// TwinCAT 3 PLC project TcoDrivesBeckhoffTests
// Title: TcoDrivesBeckhoffTests
// Company: Vortex.Library
// Author: TcOpenGroup
// ProjectVersion: 0.6.0.913
// ProgramVersion: 3.1.4024.12
// libraries:
//   Tc2_EtherCAT, * (Beckhoff Automation GmbH)
//   Tc2_MC2, * (Beckhoff Automation GmbH)
//   Tc2_Standard, * (Beckhoff Automation GmbH)
//   Tc2_System, * (Beckhoff Automation GmbH)
//   Tc3_Module, * (Beckhoff Automation GmbH)
//   TcoCore, 0.6.0.913 (Vortex.Library)
//   TcoDrivesBeckhoff, 0.6.0.913 (Vortex.Library)
// project tree:
//   GVLs/ GVL.TcGVL
//   / PlcTask1.TcTTO
//   POUs/ MAIN.TcPOU
//   Tests/TcoContext/ Sequence1Task.TcPOU, SomeTestPositions.TcPOU, SomeTestMultiPositions.TcPOU, WpfContext.TcPOU
//   Tests/TcoContext/WrappedComponent/ WrappedComponentExample.TcPOU, WrappedComponentExample_Config.TcDUT, WrappedComponentExample_Control.TcDUT, WrappedComponentExample_Status.TcDUT, WrappedComponentsExample.TcDUT
//   Tests/TcoDriveSimple/ eTcoDriveSimpleTests.TcDUT, TcoDriveSimpleTestContext.TcPOU, TcoDriveSimpleTest.TcPOU
//   Tests/TcoSingleAxis/ eTcoSingleAxisTests.TcDUT, TcoSingleAxisContext.TcPOU, TcoSingleAxisTest.TcPOU
//   Tests/TcoMultiAxis/ eTcoMultiAxisTests.TcDUT, TcoMultiAxisContext.TcPOU, TcoMultiAxisTest.TcPOU
// (motion and I/O tree: see PLC project tcodrivesbeckhoff)
// real-time tasks:
//   TASK PlcTask: cycle T#10ms, priority 20, ADS port 350
//   TASK PlcTask1: cycle T#10ms, priority 1, ADS port 351
// variable links:
//   TcoDrivesBeckhoffTests/TcoDrivesBeckhoffTests Instance <-> Device 2 (EtherCAT)/Term 1 (EK1200)/Term 12 (EL1809)
//     PlcTask1 Inputs/GVL._calibrationCam <-> Channel 1/Input
//   TcoDrivesBeckhoffTests/TcoDrivesBeckhoffTests Instance <-> NC-Task 1 SAF/Axes/Axis 1
//     PlcTask1 Inputs/GVL.Axis1.NcToPlc <-> Outputs/ToPlc
//     PlcTask1 Outputs/GVL.Axis1.PlcToNc <-> Inputs/FromPlc
//   TcoDrivesBeckhoffTests/TcoDrivesBeckhoffTests Instance <-> NC-Task 1 SAF/Axes/Axis 2
//     PlcTask1 Inputs/GVL.Axis2.NcToPlc <-> Outputs/ToPlc
//     PlcTask1 Outputs/GVL.Axis2.PlcToNc <-> Inputs/FromPlc
//   TcoDrivesBeckhoffTests/TcoDrivesBeckhoffTests Instance <-> NC-Task 1 SAF/Axes/Axis 3
//     PlcTask1 Inputs/GVL.Axis3.NcToPlc <-> Outputs/ToPlc
//     PlcTask1 Outputs/GVL.Axis3.PlcToNc <-> Inputs/FromPlc
//   TcoDrivesBeckhoffTests/TcoDrivesBeckhoffTests Instance <-> NC-Task 1 SAF/Axes/Axis 4
//     PlcTask1 Inputs/GVL.Axis4.NcToPlc <-> Outputs/ToPlc
//     PlcTask1 Outputs/GVL.Axis4.PlcToNc <-> Inputs/FromPlc

CONFIGURATION TcoDrivesBeckhoffTests
    RESOURCE PLC ON TwinCAT3
        TASK PlcTask1(INTERVAL := T#10ms, PRIORITY := 1);
        PROGRAM MAIN WITH PlcTask1 : MAIN;
    END_RESOURCE
END_CONFIGURATION

// ---- Tests/TcoContext/WrappedComponent/WrappedComponentExample_Config.TcDUT
TYPE WrappedComponentExample_Config EXTENDS TcoCore.TcoStruct :
STRUCT
    VacuumReachedStabilisation : TIME := T#100MS;
    VacuumPushTime : TIME := T#100MS;
END_STRUCT
END_TYPE

// ---- Tests/TcoContext/WrappedComponent/WrappedComponentExample_Control.TcDUT
TYPE WrappedComponentExample_Control EXTENDS TcoCore.TcoStruct :
STRUCT
    Setpoint : INT;
END_STRUCT
END_TYPE

// ---- Tests/TcoContext/WrappedComponent/WrappedComponentExample_Status.TcDUT
TYPE WrappedComponentExample_Status EXTENDS TcoCore.TcoStruct :
STRUCT
    ProgressThrow : INT;
    ActionDescription : STRING;
END_STRUCT
END_TYPE

// ---- Tests/TcoContext/WrappedComponent/WrappedComponentsExample.TcDUT
TYPE WrappedComponentsExample EXTENDS TcoCore.TcoStruct :
STRUCT
    {attribute addProperty Name "Manipulator"}
    Manipulator : TcoDrivesBeckhoff.TcoMultiAxis(THISSTRUCT);
    {attribute addProperty Name "Axis"}
    Axis : TcoDrivesBeckhoff.TcoSingleAxis(THISSTRUCT);
    {attribute addProperty Name "Drive"}
    Drive : TcoDrivesBeckhoff.TcoDriveSimple(THISSTRUCT);
END_STRUCT
END_TYPE

// ---- Tests/TcoDriveSimple/eTcoDriveSimpleTests.TcDUT
{attribute 'qualified_only'}
{attribute 'strict'}
TYPE eTcoDriveSimpleTests :
(
    Restore := 1,
    CleanUp,
    Message,
    PowerDisable,
    PowerEnable,
    Reset,
    MoveRelativePositiveWithDisabledPositiveDirection,
    MoveRelativePositiveWithEnabledPositiveDirection,
    MoveRelativeNegativeWithDisabledNegativeDirection,
    MoveRelativeNegativeWithEnabledNegativeDirection,
    HommingDirect,
    MoveVelocityPositiveWithDisabledPositiveDirection,
    MoveVelocityPositiveWithEnabledPositiveDirection,
    Stop,
    MoveVelocityNegativeWithDisabledNegativeDirection,
    MoveVelocityNegativeWithEnabledNegativeDirection,
    MoveAbsoluteDisabled,
    MoveAbsoluteDisabledPositiveDirection,
    MoveAbsoluteEnabledPositiveDirection,
    MoveAbsoluteDisabledNegativeDirection,
    MoveAbsoluteEnabledNegativeDirection,
    Last
);
END_TYPE

// ---- Tests/TcoSingleAxis/eTcoSingleAxisTests.TcDUT
{attribute 'qualified_only'}
{attribute 'strict'}
TYPE eTcoSingleAxisTests :
(
    Restore := 1,
    CleanUp,
    Message,
    PowerDisable,
    PowerEnable,
    Reset,
    MoveRelativePositiveWithDisabledPositiveDirection,
    MoveRelativePositiveWithEnabledPositiveDirection,
    MoveRelativeNegativeWithDisabledNegativeDirection,
    MoveRelativeNegativeWithEnabledNegativeDirection,
    HommingDirect,
    MoveVelocityPositiveWithDisabledPositiveDirection,
    MoveVelocityPositiveWithEnabledPositiveDirection,
    Stop,
    MoveVelocityNegativeWithDisabledNegativeDirection,
    MoveVelocityNegativeWithEnabledNegativeDirection,
    MoveAbsoluteDisabled,
    MoveAbsoluteDisabledPositiveDirection,
    MoveAbsoluteEnabledPositiveDirection,
    MoveAbsoluteDisabledNegativeDirection,
    MoveAbsoluteEnabledNegativeDirection,
    MoveAbsoluteAxisDisabled,
    MoveAbsoluteAxisDisabledPositiveDirection,
    MoveAbsoluteAxisEnabledPositiveDirection,
    MoveAbsoluteAxisDisabledNegativeDirection,
    MoveAbsoluteAxisEnabledNegativeDirection,
    MoveRelativeAxisDisabled,
    MoveRelativeAxisDisabledPositiveDirection,
    MoveRelativeAxisEnabledPositiveDirection,
    MoveRelativeAxisDisabledNegativeDirection,
    MoveRelativeAxisEnabledNegativeDirection,
    Last
);
END_TYPE

// ---- Tests/TcoMultiAxis/eTcoMultiAxisTests.TcDUT
{attribute 'qualified_only'}
{attribute 'strict'}
TYPE eTcoMultiAxisTests :
(
    Restore := 1,
    CleanUp,
    Message,
    PowerDisable,
    PowerEnable,
    Reset,
    HommingDirect,
    Stop,
    MoveAbsoluteDisabled,
    MoveAbsoluteDisabledPositiveDirection,
    MoveAbsoluteEnabledPositiveDirection,
    MoveAbsoluteDisabledNegativeDirection,
    MoveAbsoluteEnabledNegativeDirection,
    MoveAbsoluteAxisDisabled,
    MoveAbsoluteAxisDisabledPositiveDirection,
    MoveAbsoluteAxisEnabledPositiveDirection,
    MoveAbsoluteAxisDisabledNegativeDirection,
    MoveAbsoluteAxisEnabledNegativeDirection,
    MoveAbsoluteAxisDisabledPositiveDirectionAxisDisabled,
    MoveAbsoluteAxisEnabledPositiveDirectionAxisDisabled,
    MoveAbsoluteAxisDisabledNegativeDirectionAxisDisabled,
    MoveAbsoluteAxisEnabledNegativeDirectionAxisDisabled,
    Last
);
END_TYPE

// ---- GVLs/GVL.TcGVL
{attribute 'qualified_only'}
VAR_GLOBAL
    SimpleAxis1 : TcoDrivesBeckhoff.TcoAxisRef;
    SimpleAxis2 : TcoDrivesBeckhoff.TcoAxisRef;
    SingleAxis : TcoDrivesBeckhoff.TcoAxisRef;
    Axis1 : TcoDrivesBeckhoff.TcoAxisRef;
    Axis2 : TcoDrivesBeckhoff.TcoAxisRef;
    Axis3 : TcoDrivesBeckhoff.TcoAxisRef;
    Axis4 : TcoDrivesBeckhoff.TcoAxisRef;
    _calibrationCam AT %I* : BOOL;
END_VAR

// ---- POUs/MAIN.TcPOU
PROGRAM MAIN
VAR
    _tcoDriveSimpleTestContext : TcoDriveSimpleTestContext;
    _tcoSingleAxisTestContext : TcoSingleAxisContext;
    _tcoMultiAxisTestContext : TcoMultiAxisContext;
    _wpfContext : WpfContext;
    _wpfContextCall : BOOL := FALSE;
    _singleAxisTestActive : BOOL;
    _multiAxisTestActive : BOOL;
END_VAR

IF _singleAxisTestActive THEN
    _tcoSingleAxisTestContext.ProbeRun();
ELSIF _multiAxisTestActive THEN
    _tcoMultiAxisTestContext.ProbeRun();
ELSE
    _tcoDriveSimpleTestContext.ProbeRun();
END_IF

IF _wpfContextCall THEN
    _wpfContext.Run();
END_IF

END_PROGRAM

// ---- Tests/TcoDriveSimple/TcoDriveSimpleTestContext.TcPOU
FUNCTION_BLOCK TcoDriveSimpleTestContext EXTENDS TcoCore._internals_TcoContext
VAR
    _sut : TcoDriveSimpleTest(THIS^);
    _callMyPlcInstance : BOOL := FALSE;
    _enable : BOOL;
    _enablePositive : BOOL;
    _enableNegative : BOOL;
    _calibrationCam : BOOL;
    _position : LREAL;
    _velocity : LREAL;
    _acceleration : LREAL;
    _deceleration : LREAL;
    _jerk : LREAL;
    _inString : STRING;
    _done : BOOL;
    _arranged : BOOL;
    _axisReferenceType : INT;
END_VAR

METHOD PROTECTED Main
_sut(inEnable := _enable,
    inEnablePositive := _enablePositive,
    inEnableNegative := _enableNegative,
    inCalibrationCam := _calibrationCam,
    inoAxisRef := GVL.Axis1);

CASE _testId OF
    eTcoDriveSimpleTests.Restore:
        _sut.Restore();
    eTcoDriveSimpleTests.CleanUp:
        _sut._messenger.Clear();
        {region "T003_Message"}
    eTcoDriveSimpleTests.Message:
        _sut.Messenger.Error(_inString);
        _done := _plcCycleCounter > 1;
        ProbeDoneWhen(_done);
        {endregion}
        {region "T004_PowerDisable"}
    eTcoDriveSimpleTests.PowerDisable:
        _enable := FALSE;
        _done := _sut._axisStatus.Disabled; // OR _plcCycleCounter > 1;
        ProbeDoneWhen(_done);
        {endregion}
        {region "T005_PowerEnable"}
    eTcoDriveSimpleTests.PowerEnable:
        _enable := TRUE;
        _done := _sut._axisStatus.Operational; // OR _plcCycleCounter > 15;
        ProbeDoneWhen(_done);
        {endregion}
        {region "T006_Reset"}
    eTcoDriveSimpleTests.Reset:
        IF NOT _arranged THEN
            _sut.MoveRelative(inDistance := 500,
                inVelocity := 50000000,
                inAcceleration := -1,
                inDeceleration := -1,
                inJerk := -1);

            IF _sut._axisStatus.Error THEN
                _arranged := true;
            END_IF

            RETURN;
        END_IF

        _sut.Reset();
        _done := _sut.ResetTask.Done OR _sut.ResetTask.Error; // OR _plcCycleCounter > 1;
        ProbeDoneWhen(_done);
        {endregion}
        {region "T007_MoveRelativePositiveWithDisabledPositiveDirection"}
    eTcoDriveSimpleTests.MoveRelativePositiveWithDisabledPositiveDirection:
        IF NOT _arranged THEN
            _enable := TRUE;
            _enablePositive := FALSE;
            _enableNegative := FALSE;

            IF _sut._axisStatus.Operational THEN
                _arranged := TRUE;
            END_IF

            RETURN;
        END_IF;

        _sut.MoveRelative(inDistance := _position,
            inVelocity := _velocity,
            inAcceleration := _acceleration,
            inDeceleration := _deceleration,
            inJerk := _jerk);

        _done := _sut.MoveRelativeTask.Done OR _sut.MoveRelativeTask.Error; // OR _sut._axisStatus.Error;// OR _plcCycleCounter > 5;
        ProbeDoneWhen(_done);
        {endregion}
        {region "T008_MoveRelativePositiveWithEnabledPositiveDirection"}
    eTcoDriveSimpleTests.MoveRelativePositiveWithEnabledPositiveDirection:
        IF NOT _arranged THEN
            _enable := TRUE;
            _enablePositive := TRUE;
            _enableNegative := FALSE;

            IF _sut._axisStatus.Operational THEN
                _arranged := TRUE;
            END_IF

            RETURN;
        END_IF;

        _sut.MoveRelative(inDistance := _position,
            inVelocity := _velocity,
            inAcceleration := _acceleration,
            inDeceleration := _deceleration,
            inJerk := _jerk);

        _done := _sut.MoveRelativeTask.Done OR _sut.MoveRelativeTask.Error; // OR  _plcCycleCounter > 1000;
        ProbeDoneWhen(_done);
        {endregion}
        {region "T009_MoveRelativeNegativeWithDisabledNegativeDirection"}
    eTcoDriveSimpleTests.MoveRelativeNegativeWithDisabledNegativeDirection:
        IF NOT _arranged THEN
            _enable := TRUE;
            _enablePositive := FALSE;
            _enableNegative := FALSE;

            IF _sut._axisStatus.Operational THEN
                _arranged := TRUE;
            END_IF

            RETURN;
        END_IF;

        _sut.MoveRelative(inDistance := _position,
            inVelocity := _velocity,
            inAcceleration := _acceleration,
            inDeceleration := _deceleration,
            inJerk := _jerk);

        _done := _sut.MoveRelativeTask.Done OR _sut.MoveRelativeTask.Error; // OR _sut._axisStatus.Error;// OR _plcCycleCounter > 5;
        ProbeDoneWhen(_done);
        {endregion}
        {region "T010_MoveRelativeNegativeWithEnabledNegativeDirection"}
    eTcoDriveSimpleTests.MoveRelativeNegativeWithEnabledNegativeDirection:
        IF NOT _arranged THEN
            _enable := TRUE;
            _enablePositive := TRUE;
            _enableNegative := TRUE;

            IF _sut._axisStatus.Operational THEN
                _arranged := TRUE;
            END_IF

            RETURN;
        END_IF;

        _sut.MoveRelative(inDistance := _position,
            inVelocity := _velocity,
            inAcceleration := _acceleration,
            inDeceleration := _deceleration,
            inJerk := _jerk);

        _done := _sut.MoveRelativeTask.Done OR _sut.MoveRelativeTask.Error; // OR  _plcCycleCounter > 1000;
        ProbeDoneWhen(_done);
        {endregion}
        {region "T011_HommingDirect"}
    eTcoDriveSimpleTests.HommingDirect:
        IF NOT _arranged THEN
            _enable := TRUE;
            _enablePositive := FALSE;
            _enableNegative := TRUE;

            IF _sut._axisStatus.Operational THEN
                _arranged := TRUE;
            END_IF

            RETURN;
        END_IF;

        _sut.Home(inPosition := _position,
            inHomingMode := TcoDrivesBeckhoff.eHomingMode.MC_Direct,
            inClearPositionLag := FALSE,
            inSearchDirection := TcoDrivesBeckhoff.eDirection.MC_Undefined_Direction,
            inSearchVelocity := _velocity,
            inSyncDirection := TcoDrivesBeckhoff.eDirection.MC_Undefined_Direction,
            inSyncVelocity := _velocity,
            inReferenceMode := TcoDrivesBeckhoff.eEncoderReferenceMode.ENCODERREFERENCEMODE_DEFAULT);

        _done := _sut.HomeTask.Done OR _sut.HomeTask.Error; //OR _plcCycleCounter > 1000;
        ProbeDoneWhen(_done);
        {endregion}
        {region "T012_MoveVelocityPositiveWithDisabledPositiveDirection"}
    eTcoDriveSimpleTests.MoveVelocityPositiveWithDisabledPositiveDirection:
        IF NOT _arranged THEN
            _enable := TRUE;
            _enablePositive := FALSE;
            _enableNegative := FALSE;

            IF _sut._axisStatus.Operational THEN
                _arranged := TRUE;
            END_IF

            RETURN;
        END_IF;

        _sut.MoveVelocity(inVelocity := _velocity,
            inAcceleration := _acceleration,
            inDeceleration := _deceleration,
            inJerk := _jerk,
            inDirection := TcoDrivesBeckhoff.eDirection.MC_Positive_Direction);

        _done := _sut.MoveVelocityTask.Done OR _sut.MoveVelocityTask.Error; // OR  _sut._axisStatus.Error;// OR _plcCycleCounter > 5;
        ProbeDoneWhen(_done);
        {endregion}
        {region "T013_MoveVelocityPositiveWithEnabledPositiveDirection"}
    eTcoDriveSimpleTests.MoveVelocityPositiveWithEnabledPositiveDirection:
        IF NOT _arranged THEN
            _enable := TRUE;
            _enablePositive := TRUE;
            _enableNegative := FALSE;

            IF _sut._axisStatus.Operational THEN
                _arranged := TRUE;
            END_IF

            RETURN;
        END_IF;

        _sut.MoveVelocity(inVelocity := _velocity,
            inAcceleration := _acceleration,
            inDeceleration := _deceleration,
            inJerk := _jerk,
            inDirection := TcoDrivesBeckhoff.eDirection.MC_Positive_Direction);

        _done := _sut.MoveVelocityTask.Done OR _sut.MoveVelocityTask.Error; // OR  _plcCycleCounter > 1000;
        ProbeDoneWhen(_done);
        {endregion}
        {region "T014_Stop"}
    eTcoDriveSimpleTests.Stop:
        IF NOT _arranged THEN
            _enable := TRUE;
            _enablePositive := TRUE;
            _enableNegative := TRUE;

            IF _sut._axisStatus.Operational THEN
                _arranged := TRUE;
            END_IF

            RETURN;
        END_IF;

        _sut.Stop(inDeceleration := _deceleration, inJerk := _jerk);
        _done := _sut.StopTask.Done OR _sut.StopTask.Error; // OR  _plcCycleCounter > 1000;
        ProbeDoneWhen(_done);
        {endregion}
        {region "T015_MoveVelocityNegativeWithDisabledNegativeDirection"}
    eTcoDriveSimpleTests.MoveVelocityNegativeWithDisabledNegativeDirection:
        IF NOT _arranged THEN
            _enable := TRUE;
            _enablePositive := FALSE;
            _enableNegative := FALSE;

            IF _sut._axisStatus.Operational THEN
                _arranged := TRUE;
            END_IF

            RETURN;
        END_IF;

        _sut.MoveVelocity(inVelocity := _velocity,
            inAcceleration := _acceleration,
            inDeceleration := _deceleration,
            inJerk := _jerk,
            inDirection := TcoDrivesBeckhoff.eDirection.MC_Negative_Direction);

        _done := _sut.MoveVelocityTask.Done OR _sut.MoveVelocityTask.Error; // OR  _sut._axisStatus.Error;// OR _plcCycleCounter > 5;
        ProbeDoneWhen(_done);
        {endregion}
        {region "T016_MoveVelocityNegativeWithEnabledNegativeDirection"}
    eTcoDriveSimpleTests.MoveVelocityNegativeWithEnabledNegativeDirection:
        IF NOT _arranged THEN
            _enable := TRUE;
            _enablePositive := FALSE;
            _enableNegative := TRUE;

            IF _sut._axisStatus.Operational THEN
                _arranged := TRUE;
            END_IF

            RETURN;
        END_IF;

        _sut.MoveVelocity(inVelocity := _velocity,
            inAcceleration := _acceleration,
            inDeceleration := _deceleration,
            inJerk := _jerk,
            inDirection := TcoDrivesBeckhoff.eDirection.MC_Negative_Direction);

        _done := _sut.MoveVelocityTask.Done OR _sut.MoveVelocityTask.Error; // OR  _plcCycleCounter > 1000;
        ProbeDoneWhen(_done);
        {endregion}
        {region "T017_MoveAbsoluteDisabled"}
    eTcoDriveSimpleTests.MoveAbsoluteDisabled:
        IF NOT _arranged THEN
            _enable := FALSE;
            _enablePositive := FALSE;
            _enableNegative := FALSE;
            _arranged := TRUE;
            RETURN;
        END_IF;

        _sut.MoveAbsolute(inPosition := _position,
            inVelocity := _velocity,
            inAcceleration := _acceleration,
            inDeceleration := _deceleration,
            inJerk := _jerk);

        _done := _sut.MoveAbsoluteTask.Done OR _sut.MoveAbsoluteTask.Error OR _plcCycleCounter > 10;
        ProbeDoneWhen(_done);
        {endregion}
        {region "T018_MoveAbsoluteDisabledPositiveDirection"}
    eTcoDriveSimpleTests.MoveAbsoluteDisabledPositiveDirection:
        IF NOT _arranged THEN
            _enable := TRUE;
            _enablePositive := FALSE;
            _enableNegative := TRUE;
            _arranged := TRUE;
            RETURN;
        END_IF;

        _sut.MoveAbsolute(inPosition := _position,
            inVelocity := _velocity,
            inAcceleration := _acceleration,
            inDeceleration := _deceleration,
            inJerk := _jerk);

        _done := _sut.MoveAbsoluteTask.Done OR _sut.MoveAbsoluteTask.Error; // OR _sut._axisStatus.Error;// OR _plcCycleCounter > 5;
        ProbeDoneWhen(_done);
        {endregion}
        {region "T019_MoveAbsoluteEnabledPositiveDirection"}
    eTcoDriveSimpleTests.MoveAbsoluteEnabledPositiveDirection:
        IF NOT _arranged THEN
            _enable := TRUE;
            _enablePositive := TRUE;
            _enableNegative := FALSE;
            _arranged := TRUE;
            RETURN;
        END_IF;

        _sut.MoveAbsolute(inPosition := _position,
            inVelocity := _velocity,
            inAcceleration := _acceleration,
            inDeceleration := _deceleration,
            inJerk := _jerk);

        _done := _sut.MoveAbsoluteTask.Done OR _sut.MoveAbsoluteTask.Error; // OR _sut._axisStatus.Error;// OR _plcCycleCounter > 5;
        ProbeDoneWhen(_done);
        {endregion}
        {region "T020_MoveAbsoluteDisabledNegativeDirection"}
    eTcoDriveSimpleTests.MoveAbsoluteDisabledNegativeDirection:
        IF NOT _arranged THEN
            _enable := TRUE;
            _enablePositive := FALSE;
            _enableNegative := FALSE;
            _arranged := TRUE;
            RETURN;
        END_IF;

        _sut.MoveAbsolute(inPosition := _position,
            inVelocity := _velocity,
            inAcceleration := _acceleration,
            inDeceleration := _deceleration,
            inJerk := _jerk);

        _done := _sut.MoveAbsoluteTask.Done OR _sut.MoveAbsoluteTask.Error; // OR _sut._axisStatus.Error;// OR _plcCycleCounter > 5;
        ProbeDoneWhen(_done);
        {endregion}
        {region "T021_MoveAbsoluteEnabledNegativeDirection"}
    eTcoDriveSimpleTests.MoveAbsoluteEnabledNegativeDirection:
        IF NOT _arranged THEN
            _enable := TRUE;
            _enablePositive := FALSE;
            _enableNegative := TRUE;
            _arranged := TRUE;
            RETURN;
        END_IF;

        _sut.MoveAbsolute(inPosition := _position,
            inVelocity := _velocity,
            inAcceleration := _acceleration,
            inDeceleration := _deceleration,
            inJerk := _jerk);

        _done := _sut.MoveAbsoluteTask.Done OR _sut.MoveAbsoluteTask.Error; // OR _sut._axisStatus.Error;// OR _plcCycleCounter > 5;
        ProbeDoneWhen(_done);
        {endregion}
END_CASE
END_METHOD

END_FUNCTION_BLOCK

// ---- Tests/TcoDriveSimple/TcoDriveSimpleTest.TcPOU
FUNCTION_BLOCK TcoDriveSimpleTest EXTENDS TcoDrivesBeckhoff.TcoDriveSimple
VAR
    _serviceModeCount : ULINT;
    _serviceModeOverride : LREAL;
END_VAR
VAR
    _MC_ReadDriveAddress : MC_ReadDriveAddress;
    _fbEcCoeSdoRead : FB_EcCoeSdoRead;
    sNetId : T_AmsNetId;
    nSlaveAddr : UINT;
    _MotorType : STRING;
    _ftrig : Tc2_Standard.F_TRIG;
    _MC_ReadParameter : MC_ReadParameter;
END_VAR

SUPER^(inEnable := inEnable,
    inEnablePositive := inEnablePositive,
    inEnableNegative := inEnableNegative,
    inCalibrationCam := inCalibrationCam,
    inoAxisRef := inoAxisRef);

END_FUNCTION_BLOCK

// ---- Tests/TcoSingleAxis/TcoSingleAxisContext.TcPOU
FUNCTION_BLOCK TcoSingleAxisContext EXTENDS TcoCore._internals_TcoContext
VAR
    _sut : TcoSingleAxisTest(THIS^);
    _callMyPlcInstance : BOOL := FALSE;
    _enable : BOOL;
    _enablePositive : BOOL;
    _enableNegative : BOOL;
    _calibrationCam : BOOL;
    _position : LREAL;
    _velocity : LREAL;
    _acceleration : LREAL;
    _deceleration : LREAL;
    _jerk : LREAL;
    _inString : STRING;
    _done : BOOL;
    _arranged : BOOL;
    _axisReferenceType : INT;
    _positions : SomeTestPositions(THIS^);
    _moveParam : TcoSingleAxisMoveParam;
END_VAR

METHOD PROTECTED Main
_sut.Config.ErrorTime := T#1000MS;
_sut.Config.InfoTime := T#1000MS;

_sut(inEnable := _enable,
    inEnablePositive := _enablePositive,
    inEnableNegative := _enableNegative,
    inCalibrationCam := _calibrationCam,
    refAxis := GVL.Axis1,
    inoPositions := _positions);

CASE _testId OF
    eTcoSingleAxisTests.Restore:
        _sut.Restore();
    eTcoSingleAxisTests.CleanUp:
        _sut._messenger.Clear();
        {region "T003_Message"}
    eTcoSingleAxisTests.Message:
        _sut.Messenger.Error(_inString);
        _done := _plcCycleCounter > 1;
        ProbeDoneWhen(_done);
        {endregion}
        {region "T004_PowerDisable"}
    eTcoSingleAxisTests.PowerDisable:
        _enable := FALSE;
        _done := _sut.Axis._axisStatus.Disabled; // OR _plcCycleCounter > 1;
        ProbeDoneWhen(_done);
        {endregion}
        {region "T005_PowerEnable"}
    eTcoSingleAxisTests.PowerEnable:
        _enable := TRUE;
        _done := _sut.Axis._axisStatus.Operational; // OR _plcCycleCounter > 15;
        ProbeDoneWhen(_done);
        {endregion}
        {region "T006_Reset"}
    eTcoSingleAxisTests.Reset:
        IF NOT _arranged THEN
            _sut.Axis.MoveRelative(inDistance := 500,
                inVelocity := 50000000,
                inAcceleration := -1,
                inDeceleration := -1,
                inJerk := -1);

            IF _sut.Axis._axisStatus.Error THEN
                _arranged := true;
            END_IF

            RETURN;
        END_IF

        _sut.Axis.Reset();
        _done := _sut.Axis.ResetTask.Done OR _sut.Axis.ResetTask.Error; // OR _plcCycleCounter > 1;
        ProbeDoneWhen(_done);
        {endregion}
        {region "T007_MoveRelativePositiveWithDisabledPositiveDirection"}
    eTcoSingleAxisTests.MoveRelativePositiveWithDisabledPositiveDirection:
        IF NOT _arranged THEN
            _enable := TRUE;
            _enablePositive := FALSE;
            _enableNegative := FALSE;

            IF _sut.Axis._axisStatus.Operational THEN
                _arranged := TRUE;
            END_IF

            RETURN;
        END_IF;

        _sut.Axis.MoveRelative(inDistance := _position,
            inVelocity := _velocity,
            inAcceleration := _acceleration,
            inDeceleration := _deceleration,
            inJerk := _jerk);

        _done := _sut.Axis.MoveRelativeTask.Done OR _sut.Axis.MoveRelativeTask.Error; // OR _sut._axisStatus.Error;// OR _plcCycleCounter > 5;
        ProbeDoneWhen(_done);
        {endregion}
        {region "T008_MoveRelativePositiveWithEnabledPositiveDirection"}
    eTcoSingleAxisTests.MoveRelativePositiveWithEnabledPositiveDirection:
        IF NOT _arranged THEN
            _enable := TRUE;
            _enablePositive := TRUE;
            _enableNegative := FALSE;

            IF _sut.Axis._axisStatus.Operational THEN
                _arranged := TRUE;
            END_IF

            RETURN;
        END_IF;

        _sut.Axis.MoveRelative(inDistance := _position,
            inVelocity := _velocity,
            inAcceleration := _acceleration,
            inDeceleration := _deceleration,
            inJerk := _jerk);

        _done := _sut.Axis.MoveRelativeTask.Done OR _sut.Axis.MoveRelativeTask.Error; // OR  _plcCycleCounter > 1000;
        ProbeDoneWhen(_done);
        {endregion}
        {region "T009_MoveRelativeNegativeWithDisabledNegativeDirection"}
    eTcoSingleAxisTests.MoveRelativeNegativeWithDisabledNegativeDirection:
        IF NOT _arranged THEN
            _enable := TRUE;
            _enablePositive := FALSE;
            _enableNegative := FALSE;

            IF _sut.Axis._axisStatus.Operational THEN
                _arranged := TRUE;
            END_IF

            RETURN;
        END_IF;

        _sut.Axis.MoveRelative(inDistance := _position,
            inVelocity := _velocity,
            inAcceleration := _acceleration,
            inDeceleration := _deceleration,
            inJerk := _jerk);

        _done := _sut.Axis.MoveRelativeTask.Done OR _sut.Axis.MoveRelativeTask.Error; // OR _sut._axisStatus.Error;// OR _plcCycleCounter > 5;
        ProbeDoneWhen(_done);
        {endregion}
        {region "T010_MoveRelativeNegativeWithEnabledNegativeDirection"}
    eTcoSingleAxisTests.MoveRelativeNegativeWithEnabledNegativeDirection:
        IF NOT _arranged THEN
            _enable := TRUE;
            _enablePositive := TRUE;
            _enableNegative := TRUE;

            IF _sut.Axis._axisStatus.Operational THEN
                _arranged := TRUE;
            END_IF

            RETURN;
        END_IF;

        _sut.Axis.MoveRelative(inDistance := _position,
            inVelocity := _velocity,
            inAcceleration := _acceleration,
            inDeceleration := _deceleration,
            inJerk := _jerk);

        _done := _sut.Axis.MoveRelativeTask.Done OR _sut.Axis.MoveRelativeTask.Error; // OR  _plcCycleCounter > 1000;
        ProbeDoneWhen(_done);
        {endregion}
        {region "T011_HommingDirect"}
    eTcoSingleAxisTests.HommingDirect:
        IF NOT _arranged THEN
            _enable := TRUE;
            _enablePositive := FALSE;
            _enableNegative := TRUE;

            IF _sut.Axis._axisStatus.Operational THEN
                _arranged := TRUE;
            END_IF

            RETURN;
        END_IF;

        _sut.Axis.Home(inPosition := _position,
            inHomingMode := TcoDrivesBeckhoff.eHomingMode.MC_Direct,
            inClearPositionLag := FALSE,
            inSearchDirection := TcoDrivesBeckhoff.eDirection.MC_Undefined_Direction,
            inSearchVelocity := _velocity,
            inSyncDirection := TcoDrivesBeckhoff.eDirection.MC_Undefined_Direction,
            inSyncVelocity := _velocity,
            inReferenceMode := TcoDrivesBeckhoff.eEncoderReferenceMode.ENCODERREFERENCEMODE_DEFAULT);

        _done := _sut.Axis.HomeTask.Done OR _sut.Axis.HomeTask.Error; //OR _plcCycleCounter > 1000;
        ProbeDoneWhen(_done);
        {endregion}
        {region "T012_MoveVelocityPositiveWithDisabledPositiveDirection"}
    eTcoSingleAxisTests.MoveVelocityPositiveWithDisabledPositiveDirection:
        IF NOT _arranged THEN
            _enable := TRUE;
            _enablePositive := FALSE;
            _enableNegative := FALSE;

            IF _sut.Axis._axisStatus.Operational THEN
                _arranged := TRUE;
            END_IF

            RETURN;
        END_IF;

        _sut.Axis.MoveVelocity(inVelocity := _velocity,
            inAcceleration := _acceleration,
            inDeceleration := _deceleration,
            inJerk := _jerk,
            inDirection := TcoDrivesBeckhoff.eDirection.MC_Positive_Direction);

        _done := _sut.Axis.MoveVelocityTask.Done OR _sut.Axis.MoveVelocityTask.Error; // OR  _sut._axisStatus.Error;// OR _plcCycleCounter > 5;
        ProbeDoneWhen(_done);
        {endregion}
        {region "T013_MoveVelocityPositiveWithEnabledPositiveDirection"}
    eTcoSingleAxisTests.MoveVelocityPositiveWithEnabledPositiveDirection:
        IF NOT _arranged THEN
            _enable := TRUE;
            _enablePositive := TRUE;
            _enableNegative := FALSE;

            IF _sut.Axis._axisStatus.Operational THEN
                _arranged := TRUE;
            END_IF

            RETURN;
        END_IF;

        _sut.Axis.MoveVelocity(inVelocity := _velocity,
            inAcceleration := _acceleration,
            inDeceleration := _deceleration,
            inJerk := _jerk,
            inDirection := TcoDrivesBeckhoff.eDirection.MC_Positive_Direction);

        _done := _sut.Axis.MoveVelocityTask.Done OR _sut.Axis.MoveVelocityTask.Error; // OR  _plcCycleCounter > 1000;
        ProbeDoneWhen(_done);
        {endregion}
        {region "T014_Stop"}
    eTcoSingleAxisTests.Stop:
        IF NOT _arranged THEN
            _enable := TRUE;
            _enablePositive := TRUE;
            _enableNegative := TRUE;

            IF _sut.Axis._axisStatus.Operational THEN
                _arranged := TRUE;
            END_IF

            RETURN;
        END_IF;

        _sut.Axis.Stop(inDeceleration := _deceleration, inJerk := _jerk);
        _done := _sut.Axis.StopTask.Done OR _sut.Axis.StopTask.Error; // OR  _plcCycleCounter > 1000;
        ProbeDoneWhen(_done);
        {endregion}
        {region "T015_MoveVelocityNegativeWithDisabledNegativeDirection"}
    eTcoSingleAxisTests.MoveVelocityNegativeWithDisabledNegativeDirection:
        IF NOT _arranged THEN
            _enable := TRUE;
            _enablePositive := FALSE;
            _enableNegative := FALSE;

            IF _sut.Axis._axisStatus.Operational THEN
                _arranged := TRUE;
            END_IF

            RETURN;
        END_IF;

        _sut.Axis.MoveVelocity(inVelocity := _velocity,
            inAcceleration := _acceleration,
            inDeceleration := _deceleration,
            inJerk := _jerk,
            inDirection := TcoDrivesBeckhoff.eDirection.MC_Negative_Direction);

        _done := _sut.Axis.MoveVelocityTask.Done OR _sut.Axis.MoveVelocityTask.Error; // OR  _sut._axisStatus.Error;// OR _plcCycleCounter > 5;
        ProbeDoneWhen(_done);
        {endregion}
        {region "T016_MoveVelocityNegativeWithEnabledNegativeDirection"}
    eTcoSingleAxisTests.MoveVelocityNegativeWithEnabledNegativeDirection:
        IF NOT _arranged THEN
            _enable := TRUE;
            _enablePositive := FALSE;
            _enableNegative := TRUE;

            IF _sut.Axis._axisStatus.Operational THEN
                _arranged := TRUE;
            END_IF

            RETURN;
        END_IF;

        _sut.Axis.MoveVelocity(inVelocity := _velocity,
            inAcceleration := _acceleration,
            inDeceleration := _deceleration,
            inJerk := _jerk,
            inDirection := TcoDrivesBeckhoff.eDirection.MC_Negative_Direction);

        _done := _sut.Axis.MoveVelocityTask.Done OR _sut.Axis.MoveVelocityTask.Error; // OR  _plcCycleCounter > 1000;
        ProbeDoneWhen(_done);
        {endregion}
        {region "T017_MoveAbsoluteDisabled"}
    eTcoSingleAxisTests.MoveAbsoluteDisabled:
        IF NOT _arranged THEN
            _enable := FALSE;
            _enablePositive := FALSE;
            _enableNegative := FALSE;
            _arranged := TRUE;
            RETURN;
        END_IF;

        _sut.Axis.MoveAbsolute(inPosition := _position,
            inVelocity := _velocity,
            inAcceleration := _acceleration,
            inDeceleration := _deceleration,
            inJerk := _jerk);

        _done := _sut.Axis.MoveAbsoluteTask.Done OR _sut.Axis.MoveAbsoluteTask.Error OR _plcCycleCounter > 10;
        ProbeDoneWhen(_done);
        {endregion}
        {region "T018_MoveAbsoluteDisabledPositiveDirection"}
    eTcoSingleAxisTests.MoveAbsoluteDisabledPositiveDirection:
        IF NOT _arranged THEN
            _enable := TRUE;
            _enablePositive := FALSE;
            _enableNegative := TRUE;
            _arranged := TRUE;
            RETURN;
        END_IF;

        _sut.Axis.MoveAbsolute(inPosition := _position,
            inVelocity := _velocity,
            inAcceleration := _acceleration,
            inDeceleration := _deceleration,
            inJerk := _jerk);

        _done := _sut.Axis.MoveAbsoluteTask.Done OR _sut.Axis.MoveAbsoluteTask.Error; // OR _sut._axisStatus.Error;// OR _plcCycleCounter > 5;
        ProbeDoneWhen(_done);
        {endregion}
        {region "T019_MoveAbsoluteEnabledPositiveDirection"}
    eTcoSingleAxisTests.MoveAbsoluteEnabledPositiveDirection:
        IF NOT _arranged THEN
            _enable := TRUE;
            _enablePositive := TRUE;
            _enableNegative := FALSE;
            _arranged := TRUE;
            RETURN;
        END_IF;

        _sut.Axis.MoveAbsolute(inPosition := _position,
            inVelocity := _velocity,
            inAcceleration := _acceleration,
            inDeceleration := _deceleration,
            inJerk := _jerk);

        _done := _sut.Axis.MoveAbsoluteTask.Done OR _sut.Axis.MoveAbsoluteTask.Error; // OR _sut._axisStatus.Error;// OR _plcCycleCounter > 5;
        ProbeDoneWhen(_done);
        {endregion}
        {region "T020_MoveAbsoluteDisabledNegativeDirection"}
    eTcoSingleAxisTests.MoveAbsoluteDisabledNegativeDirection:
        IF NOT _arranged THEN
            _enable := TRUE;
            _enablePositive := FALSE;
            _enableNegative := FALSE;
            _arranged := TRUE;
            RETURN;
        END_IF;

        _sut.Axis.MoveAbsolute(inPosition := _position,
            inVelocity := _velocity,
            inAcceleration := _acceleration,
            inDeceleration := _deceleration,
            inJerk := _jerk);

        _done := _sut.Axis.MoveAbsoluteTask.Done OR _sut.Axis.MoveAbsoluteTask.Error; // OR _sut._axisStatus.Error;// OR _plcCycleCounter > 5;
        ProbeDoneWhen(_done);
        {endregion}
        {region "T021_MoveAbsoluteEnabledNegativeDirection"}
    eTcoSingleAxisTests.MoveAbsoluteEnabledNegativeDirection:
        IF NOT _arranged THEN
            _enable := TRUE;
            _enablePositive := FALSE;
            _enableNegative := TRUE;
            _arranged := TRUE;
            RETURN;
        END_IF;

        _sut.Axis.MoveAbsolute(inPosition := _position,
            inVelocity := _velocity,
            inAcceleration := _acceleration,
            inDeceleration := _deceleration,
            inJerk := _jerk);

        _done := _sut.Axis.MoveAbsoluteTask.Done OR _sut.MoveAbsoluteTask.Error; // OR _sut._axisStatus.Error;// OR _plcCycleCounter > 5;
        ProbeDoneWhen(_done);
        {endregion}
        {region "T022_MoveAbsoluteAxisDisabled"}
    eTcoSingleAxisTests.MoveAbsoluteAxisDisabled:
        IF NOT _arranged THEN
            _sut.Restore();
            _enable := FALSE;
            _enablePositive := FALSE;
            _enableNegative := FALSE;
            _arranged := TRUE;
            RETURN;
        END_IF;

        _moveParam.Position := _position;
        _moveParam.Velocity := _velocity;
        _moveParam.Acceleration := _acceleration;
        _moveParam.Deceleration := _deceleration;
        _moveParam.Jerk := _jerk;
        _sut.MoveAbsolute(_moveParam);
        _done := _sut.MoveAbsoluteTask.Done OR (_sut.Axis.MoveAbsoluteTask.Error AND _sut.MoveAbsoluteTask.Error) OR _plcCycleCounter > 10;
        ProbeDoneWhen(_done);
        {endregion}
        {region "T023_MoveAbsoluteAxisDisabledPositiveDirection"}
    eTcoSingleAxisTests.MoveAbsoluteAxisDisabledPositiveDirection:
        IF NOT _arranged THEN
            _sut.Restore();
            _enable := TRUE;
            _enablePositive := FALSE;
            _enableNegative := TRUE;
            _arranged := TRUE;
            RETURN;
        END_IF;

        _moveParam.Position := _position;
        _moveParam.Velocity := _velocity;
        _moveParam.Acceleration := _acceleration;
        _moveParam.Deceleration := _deceleration;
        _moveParam.Jerk := _jerk;
        _sut.MoveAbsolute(_moveParam);
        _done := _sut.MoveAbsoluteTask.Done OR (_sut.Axis.MoveAbsoluteTask.Error AND _sut.MoveAbsoluteTask.Error);
        ProbeDoneWhen(_done);
        {endregion}
        {region "T024_MoveAbsoluteAxisEnabledPositiveDirection"}
    eTcoSingleAxisTests.MoveAbsoluteAxisEnabledPositiveDirection:
        IF NOT _arranged THEN
            _sut.Restore();
            _enable := TRUE;
            _enablePositive := TRUE;
            _enableNegative := FALSE;
            _arranged := TRUE;
            RETURN;
        END_IF;

        _moveParam.Position := _position;
        _moveParam.Velocity := _velocity;
        _moveParam.Acceleration := _acceleration;
        _moveParam.Deceleration := _deceleration;
        _moveParam.Jerk := _jerk;
        _sut.MoveAbsolute(_moveParam);
        _done := _sut.MoveAbsoluteTask.Done OR (_sut.Axis.MoveAbsoluteTask.Error AND _sut.MoveAbsoluteTask.Error);
        ProbeDoneWhen(_done);
        {endregion}
        {region "T025_MoveAbsoluteAxisDisabledNegativeDirection"}
    eTcoSingleAxisTests.MoveAbsoluteAxisDisabledNegativeDirection:
        IF NOT _arranged THEN
            _sut.Restore();
            _enable := TRUE;
            _enablePositive := FALSE;
            _enableNegative := FALSE;
            _arranged := TRUE;
            RETURN;
        END_IF;

        _moveParam.Position := _position;
        _moveParam.Velocity := _velocity;
        _moveParam.Acceleration := _acceleration;
        _moveParam.Deceleration := _deceleration;
        _moveParam.Jerk := _jerk;
        _sut.MoveAbsolute(_moveParam);
        _done := _sut.MoveAbsoluteTask.Done OR (_sut.Axis.MoveAbsoluteTask.Error AND _sut.MoveAbsoluteTask.Error);
        ProbeDoneWhen(_done);
        {endregion}
        {region "T026_MoveAbsoluteAxisEnabledNegativeDirection"}
    eTcoSingleAxisTests.MoveAbsoluteAxisEnabledNegativeDirection:
        IF NOT _arranged THEN
            _sut.Restore();
            _enable := TRUE;
            _enablePositive := FALSE;
            _enableNegative := TRUE;
            _arranged := TRUE;
            RETURN;
        END_IF;

        _moveParam.Position := _position;
        _moveParam.Velocity := _velocity;
        _moveParam.Acceleration := _acceleration;
        _moveParam.Deceleration := _deceleration;
        _moveParam.Jerk := _jerk;
        _sut.MoveAbsolute(_moveParam);
        _done := _sut.MoveAbsoluteTask.Done OR (_sut.MoveAbsoluteTask.Error AND _sut.MoveAbsoluteTask.Error);
        ProbeDoneWhen(_done);
        {endregion}
        {region "T027_MoveRelativeAxisDisabled"}
    eTcoSingleAxisTests.MoveRelativeAxisDisabled:
        IF NOT _arranged THEN
            _sut.Restore();
            _enable := FALSE;
            _enablePositive := FALSE;
            _enableNegative := FALSE;
            _arranged := TRUE;
            RETURN;
        END_IF;

        _moveParam.Position := _position;
        _moveParam.Velocity := _velocity;
        _moveParam.Acceleration := _acceleration;
        _moveParam.Deceleration := _deceleration;
        _moveParam.Jerk := _jerk;
        _sut.MoveRelative(_moveParam);
        _done := _sut.MoveRelativeTask.Done OR (_sut.Axis.MoveRelativeTask.Error AND _sut.MoveRelativeTask.Error) OR _plcCycleCounter > 10;
        ProbeDoneWhen(_done);
        {endregion}
        {region "T028_MoveRelativeAxisDisabledPositiveDirection"}
    eTcoSingleAxisTests.MoveRelativeAxisDisabledPositiveDirection:
        IF NOT _arranged THEN
            _sut.Restore();
            _enable := TRUE;
            _enablePositive := FALSE;
            _enableNegative := TRUE;
            _arranged := TRUE;
            RETURN;
        END_IF;

        _moveParam.Position := _position;
        _moveParam.Velocity := _velocity;
        _moveParam.Acceleration := _acceleration;
        _moveParam.Deceleration := _deceleration;
        _moveParam.Jerk := _jerk;
        _sut.MoveRelative(_moveParam);
        _done := _sut.MoveRelativeTask.Done OR (_sut.Axis.MoveRelativeTask.Error AND _sut.MoveRelativeTask.Error);
        ProbeDoneWhen(_done);
        {endregion}
        {region "T029_MoveRelativeAxisEnabledPositiveDirection"}
    eTcoSingleAxisTests.MoveRelativeAxisEnabledPositiveDirection:
        IF NOT _arranged THEN
            _sut.Restore();
            _enable := TRUE;
            _enablePositive := TRUE;
            _enableNegative := FALSE;
            _arranged := TRUE;
            RETURN;
        END_IF;

        _moveParam.Position := _position;
        _moveParam.Velocity := _velocity;
        _moveParam.Acceleration := _acceleration;
        _moveParam.Deceleration := _deceleration;
        _moveParam.Jerk := _jerk;
        _sut.MoveRelative(_moveParam);
        _done := _sut.MoveRelativeTask.Done OR (_sut.Axis.MoveRelativeTask.Error AND _sut.MoveRelativeTask.Error);
        ProbeDoneWhen(_done);
        {endregion}
        {region "T030_MoveRelativeAxisDisabledNegativeDirection"}
    eTcoSingleAxisTests.MoveRelativeAxisDisabledNegativeDirection:
        IF NOT _arranged THEN
            _sut.Restore();
            _enable := TRUE;
            _enablePositive := FALSE;
            _enableNegative := FALSE;
            _arranged := TRUE;
            RETURN;
        END_IF;

        _moveParam.Position := _position;
        _moveParam.Velocity := _velocity;
        _moveParam.Acceleration := _acceleration;
        _moveParam.Deceleration := _deceleration;
        _moveParam.Jerk := _jerk;
        _sut.MoveRelative(_moveParam);
        _done := _sut.MoveRelativeTask.Done OR (_sut.Axis.MoveRelativeTask.Error AND _sut.MoveRelativeTask.Error);
        ProbeDoneWhen(_done);
        {endregion}
        {region "T031_MoveRelativeAxisEnabledNegativeDirection"}
    eTcoSingleAxisTests.MoveRelativeAxisEnabledNegativeDirection:
        IF NOT _arranged THEN
            _sut.Restore();
            _enable := TRUE;
            _enablePositive := FALSE;
            _enableNegative := TRUE;
            _arranged := TRUE;
            RETURN;
        END_IF;

        _moveParam.Position := _position;
        _moveParam.Velocity := _velocity;
        _moveParam.Acceleration := _acceleration;
        _moveParam.Deceleration := _deceleration;
        _moveParam.Jerk := _jerk;
        _sut.MoveRelative(_moveParam);
        _done := _sut.MoveRelativeTask.Done OR (_sut.MoveRelativeTask.Error AND _sut.MoveRelativeTask.Error);
        ProbeDoneWhen(_done);
        {endregion}
END_CASE
END_METHOD

END_FUNCTION_BLOCK

// ---- Tests/TcoSingleAxis/TcoSingleAxisTest.TcPOU
FUNCTION_BLOCK TcoSingleAxisTest EXTENDS TcoDrivesBeckhoff.TcoSingleAxis
VAR
    _serviceModeCount : ULINT;
    _serviceModeOverride : LREAL;
    inoPosition : TcoSingleAxisPositionsRootContainer(THIS^);
END_VAR
VAR
    _MC_ReadDriveAddress : MC_ReadDriveAddress;
    _fbEcCoeSdoRead : FB_EcCoeSdoRead;
    sNetId : T_AmsNetId;
    nSlaveAddr : UINT;
    _MotorType : STRING;
    _ftrig : Tc2_Standard.F_TRIG;
    _MC_ReadParameter : MC_ReadParameter;
END_VAR

SUPER^(inEnable := inEnable,
    inEnablePositive := inEnablePositive,
    inEnableNegative := inEnableNegative,
    inCalibrationCam := inCalibrationCam,
    refAxis := refAxis,
    inoPositions := inoPosition);

END_FUNCTION_BLOCK

// ---- Tests/TcoContext/SomeTestPositions.TcPOU
FUNCTION_BLOCK SomeTestPositions EXTENDS TcoDrivesBeckhoff.TcoSingleAxisPositionsRootContainer
VAR_INPUT
END_VAR
VAR_OUTPUT
END_VAR
VAR
    {attribute addProperty Name "<#Pick Position#>"}
    PickPosition : TcoDrivesBeckhoff.TcoMultiAxisMoveParam;
    {attribute addProperty Name "<#Place  Position#>"}
    PlacePosition : TcoDrivesBeckhoff.TcoMultiAxisMoveParam;
END_VAR

END_FUNCTION_BLOCK

// ---- Tests/TcoMultiAxis/TcoMultiAxisContext.TcPOU
FUNCTION_BLOCK TcoMultiAxisContext EXTENDS TcoCore._internals_TcoContext
VAR
    _sut : TcoMultiAxisTest(THIS^);
    _callMyPlcInstance : BOOL := FALSE;
    _enable : BOOL;
    _enablePositive : BOOL;
    _enableNegative : BOOL;
    _calibrationCam : BOOL;
    _positionAxis1 : LREAL;
    _positionAxis2 : LREAL;
    _positionAxis3 : LREAL;
    _positionAxis4 : LREAL;
    _velocity : LREAL;
    _acceleration : LREAL;
    _deceleration : LREAL;
    _jerk : LREAL;
    _inString : STRING;
    _done : BOOL;
    _arranged : BOOL;
    _axis1Disabled : BOOL;
    _axis2Disabled : BOOL;
    _axis3Disabled : BOOL;
    _axis4Disabled : BOOL;
    _axisReferenceType : INT;
    _positions : SomeTestMultiPositions(THIS^);
    _moveParam : TcoMultiAxisMoveParam;
END_VAR

METHOD PROTECTED Main
_sut.Config.ErrorTime := T#1000MS;
_sut.Config.InfoTime := T#1000MS;
_sut.Config.Axis1Disabled := _axis1Disabled;
_sut.Config.Axis2Disabled := _axis2Disabled;
_sut.Config.Axis3Disabled := _axis3Disabled;
_sut.Config.Axis4Disabled := _axis4Disabled;

_sut(inEnableAxis1 := _enable,
    inEnablePositiveAxis1 := _enablePositive,
    inEnableNegativeAxis1 := _enableNegative,
    inCalibrationCamAxis1 := _calibrationCam,
    refAxis1 := GVL.Axis1,
    inEnableAxis2 := _enable,
    inEnablePositiveAxis2 := _enablePositive,
    inEnableNegativeAxis2 := _enableNegative,
    inCalibrationCamAxis2 := _calibrationCam,
    refAxis2 := GVL.Axis2,
    inEnableAxis3 := _enable,
    inEnablePositiveAxis3 := _enablePositive,
    inEnableNegativeAxis3 := _enableNegative,
    inCalibrationCamAxis3 := _calibrationCam,
    refAxis3 := GVL.Axis3,
    inEnableAxis4 := _enable,
    inEnablePositiveAxis4 := _enablePositive,
    inEnableNegativeAxis4 := _enableNegative,
    inCalibrationCamAxis4 := _calibrationCam,
    refAxis4 := GVL.Axis4,
    inoPositions := _positions);

CASE _testId OF
    eTcoMultiAxisTests.Restore:
        _axis1Disabled := false;
        _axis2Disabled := FALSE;
        _axis3Disabled := FALSE;
        _axis4Disabled := FALSE;
        _sut.Restore();
    eTcoMultiAxisTests.CleanUp:
        _sut._messenger.Clear();
        _sut.ResetDrivesTask.Restore();
        _sut.SoeResetDrivesTask.Restore();
        _sut.MoveAbsoluteTask.Restore();
        _sut.AbortTask.Restore();
        {region "T003_Message"}
    eTcoMultiAxisTests.Message:
        _sut.Messenger.Error(_inString);
        _done := _plcCycleCounter > 1;
        ProbeDoneWhen(_done);
        {endregion}
        {region "T004_PowerDisable"}
    eTcoMultiAxisTests.PowerDisable:
        _enable := FALSE;

        _done := _sut.Axis_1._axisStatus.Disabled AND
            _sut.Axis_2._axisStatus.Disabled AND
            _sut.Axis_3._axisStatus.Disabled AND
            _sut.Axis_4._axisStatus.Disabled;

        ProbeDoneWhen(_done);
        {endregion}
        {region "T005_PowerEnable"}
    eTcoMultiAxisTests.PowerEnable:
        _enable := TRUE;

        _done := _sut.Axis_1._axisStatus.StandStill AND
            _sut.Axis_2._axisStatus.StandStill AND
            _sut.Axis_3._axisStatus.StandStill AND
            _sut.Axis_4._axisStatus.StandStill;

        ProbeDoneWhen(_done);
        {endregion}
        {region "T006_Reset"}
    eTcoMultiAxisTests.Reset:
        IF NOT _arranged THEN
            _sut.Axis_1.MoveRelative(inDistance := 500,
                inVelocity := 50000000,
                inAcceleration := -1,
                inDeceleration := -1,
                inJerk := -1);

            _sut.Axis_2.MoveRelative(inDistance := 500,
                inVelocity := 50000000,
                inAcceleration := -1,
                inDeceleration := -1,
                inJerk := -1);

            _sut.Axis_3.MoveRelative(inDistance := 500,
                inVelocity := 50000000,
                inAcceleration := -1,
                inDeceleration := -1,
                inJerk := -1);

            _sut.Axis_4.MoveRelative(inDistance := 500,
                inVelocity := 50000000,
                inAcceleration := -1,
                inDeceleration := -1,
                inJerk := -1);

            IF _sut.Axis_1._axisStatus.Error OR _sut.Axis_2._axisStatus.Error OR _sut.Axis_3._axisStatus.Error OR _sut.Axis_4._axisStatus.Error THEN
                _arranged := TRUE;
            END_IF

            RETURN;
        END_IF

        _sut.ResetDrives();
        _done := _sut.ResetDrivesTask.Done;
        ProbeDoneWhen(_done);
        {endregion}
        {region "T011_HommingDirect"}
    eTcoMultiAxisTests.HommingDirect:
        IF NOT _arranged THEN
            _enable := TRUE;
            _enablePositive := TRUE;
            _enableNegative := TRUE;

            IF _sut.Axis_1._axisStatus.Operational AND
                _sut.Axis_2._axisStatus.Operational AND
                _sut.Axis_3._axisStatus.Operational AND
                _sut.Axis_4._axisStatus.Operational THEN
                _arranged := TRUE;
            END_IF

            RETURN;
        END_IF;

        _sut.Axis_1.Home(inPosition := _positionAxis1,
            inHomingMode := TcoDrivesBeckhoff.eHomingMode.MC_Direct,
            inClearPositionLag := FALSE,
            inSearchDirection := TcoDrivesBeckhoff.eDirection.MC_Undefined_Direction,
            inSearchVelocity := _velocity,
            inSyncDirection := TcoDrivesBeckhoff.eDirection.MC_Undefined_Direction,
            inSyncVelocity := _velocity,
            inReferenceMode := TcoDrivesBeckhoff.eEncoderReferenceMode.ENCODERREFERENCEMODE_DEFAULT);

        _sut.Axis_2.Home(inPosition := _positionAxis2,
            inHomingMode := TcoDrivesBeckhoff.eHomingMode.MC_Direct,
            inClearPositionLag := FALSE,
            inSearchDirection := TcoDrivesBeckhoff.eDirection.MC_Undefined_Direction,
            inSearchVelocity := _velocity,
            inSyncDirection := TcoDrivesBeckhoff.eDirection.MC_Undefined_Direction,
            inSyncVelocity := _velocity,
            inReferenceMode := TcoDrivesBeckhoff.eEncoderReferenceMode.ENCODERREFERENCEMODE_DEFAULT);

        _sut.Axis_3.Home(inPosition := _positionAxis3,
            inHomingMode := TcoDrivesBeckhoff.eHomingMode.MC_Direct,
            inClearPositionLag := FALSE,
            inSearchDirection := TcoDrivesBeckhoff.eDirection.MC_Undefined_Direction,
            inSearchVelocity := _velocity,
            inSyncDirection := TcoDrivesBeckhoff.eDirection.MC_Undefined_Direction,
            inSyncVelocity := _velocity,
            inReferenceMode := TcoDrivesBeckhoff.eEncoderReferenceMode.ENCODERREFERENCEMODE_DEFAULT);

        _sut.Axis_4.Home(inPosition := _positionAxis4,
            inHomingMode := TcoDrivesBeckhoff.eHomingMode.MC_Direct,
            inClearPositionLag := FALSE,
            inSearchDirection := TcoDrivesBeckhoff.eDirection.MC_Undefined_Direction,
            inSearchVelocity := _velocity,
            inSyncDirection := TcoDrivesBeckhoff.eDirection.MC_Undefined_Direction,
            inSyncVelocity := _velocity,
            inReferenceMode := TcoDrivesBeckhoff.eEncoderReferenceMode.ENCODERREFERENCEMODE_DEFAULT);

        _done := (_sut.Axis_1.HomeTask.Done OR _sut.Axis_1.HomeTask.Error) AND
            (_sut.Axis_2.HomeTask.Done OR _sut.Axis_2.HomeTask.Error) AND
            (_sut.Axis_3.HomeTask.Done OR _sut.Axis_3.HomeTask.Error) AND
            (_sut.Axis_4.HomeTask.Done OR _sut.Axis_4.HomeTask.Error);

        ProbeDoneWhen(_done);
        {endregion}
        {region "T017_MoveAbsoluteDisabled"}
    eTcoMultiAxisTests.MoveAbsoluteDisabled:
        IF NOT _arranged THEN
            _enable := FALSE;
            _enablePositive := FALSE;
            _enableNegative := FALSE;
            _arranged := TRUE;
            RETURN;
        END_IF;

        _sut.Axis_1.MoveAbsolute(inPosition := _positionAxis1,
            inVelocity := _velocity,
            inAcceleration := _acceleration,
            inDeceleration := _deceleration,
            inJerk := _jerk);

        _sut.Axis_2.MoveAbsolute(inPosition := _positionAxis2,
            inVelocity := _velocity,
            inAcceleration := _acceleration,
            inDeceleration := _deceleration,
            inJerk := _jerk);

        _sut.Axis_3.MoveAbsolute(inPosition := _positionAxis3,
            inVelocity := _velocity,
            inAcceleration := _acceleration,
            inDeceleration := _deceleration,
            inJerk := _jerk);

        _sut.Axis_4.MoveAbsolute(inPosition := _positionAxis4,
            inVelocity := _velocity,
            inAcceleration := _acceleration,
            inDeceleration := _deceleration,
            inJerk := _jerk);

        _done := (_sut.Axis_1.MoveAbsoluteTask.Done OR _sut.Axis_1.MoveAbsoluteTask.Error OR _plcCycleCounter > 10) AND
            (_sut.Axis_2.MoveAbsoluteTask.Done OR _sut.Axis_2.MoveAbsoluteTask.Error OR _plcCycleCounter > 10) AND
            (_sut.Axis_3.MoveAbsoluteTask.Done OR _sut.Axis_3.MoveAbsoluteTask.Error OR _plcCycleCounter > 10) AND
            (_sut.Axis_4.MoveAbsoluteTask.Done OR _sut.Axis_4.MoveAbsoluteTask.Error OR _plcCycleCounter > 10);

        ProbeDoneWhen(_done);
        {endregion}
        {region "T018_MoveAbsoluteDisabledPositiveDirection"}
    eTcoMultiAxisTests.MoveAbsoluteDisabledPositiveDirection:
        IF NOT _arranged THEN
            _enable := TRUE;
            _enablePositive := FALSE;
            _enableNegative := TRUE;
            _arranged := TRUE;
            RETURN;
        END_IF;

        _sut.Axis_1.MoveAbsolute(inPosition := _positionAxis1,
            inVelocity := _velocity,
            inAcceleration := _acceleration,
            inDeceleration := _deceleration,
            inJerk := _jerk);

        _sut.Axis_2.MoveAbsolute(inPosition := _positionAxis2,
            inVelocity := _velocity,
            inAcceleration := _acceleration,
            inDeceleration := _deceleration,
            inJerk := _jerk);

        _sut.Axis_3.MoveAbsolute(inPosition := _positionAxis3,
            inVelocity := _velocity,
            inAcceleration := _acceleration,
            inDeceleration := _deceleration,
            inJerk := _jerk);

        _sut.Axis_4.MoveAbsolute(inPosition := _positionAxis4,
            inVelocity := _velocity,
            inAcceleration := _acceleration,
            inDeceleration := _deceleration,
            inJerk := _jerk);

        _done := (_sut.Axis_1.MoveAbsoluteTask.Done OR _sut.Axis_1.MoveAbsoluteTask.Error) AND
            (_sut.Axis_2.MoveAbsoluteTask.Done OR _sut.Axis_2.MoveAbsoluteTask.Error) AND
            (_sut.Axis_3.MoveAbsoluteTask.Done OR _sut.Axis_3.MoveAbsoluteTask.Error) AND
            (_sut.Axis_4.MoveAbsoluteTask.Done OR _sut.Axis_4.MoveAbsoluteTask.Error);

        ProbeDoneWhen(_done);
        {endregion}
        {region "T019_MoveAbsoluteEnabledPositiveDirection"}
    eTcoMultiAxisTests.MoveAbsoluteEnabledPositiveDirection:
        IF NOT _arranged THEN
            _enable := TRUE;
            _enablePositive := TRUE;
            _enableNegative := FALSE;
            _arranged := TRUE;
            RETURN;
        END_IF;

        _sut.Axis_1.MoveAbsolute(inPosition := _positionAxis1,
            inVelocity := _velocity,
            inAcceleration := _acceleration,
            inDeceleration := _deceleration,
            inJerk := _jerk);

        _sut.Axis_2.MoveAbsolute(inPosition := _positionAxis2,
            inVelocity := _velocity,
            inAcceleration := _acceleration,
            inDeceleration := _deceleration,
            inJerk := _jerk);

        _sut.Axis_3.MoveAbsolute(inPosition := _positionAxis3,
            inVelocity := _velocity,
            inAcceleration := _acceleration,
            inDeceleration := _deceleration,
            inJerk := _jerk);

        _sut.Axis_4.MoveAbsolute(inPosition := _positionAxis4,
            inVelocity := _velocity,
            inAcceleration := _acceleration,
            inDeceleration := _deceleration,
            inJerk := _jerk);

        _done := (_sut.Axis_1.MoveAbsoluteTask.Done OR _sut.Axis_1.MoveAbsoluteTask.Error) AND
            (_sut.Axis_2.MoveAbsoluteTask.Done OR _sut.Axis_2.MoveAbsoluteTask.Error) AND
            (_sut.Axis_3.MoveAbsoluteTask.Done OR _sut.Axis_3.MoveAbsoluteTask.Error) AND
            (_sut.Axis_4.MoveAbsoluteTask.Done OR _sut.Axis_4.MoveAbsoluteTask.Error);

        ProbeDoneWhen(_done);
        {endregion}
        {region "T020_MoveAbsoluteDisabledNegativeDirection"}
    eTcoMultiAxisTests.MoveAbsoluteDisabledNegativeDirection:
        IF NOT _arranged THEN
            _enable := TRUE;
            _enablePositive := FALSE;
            _enableNegative := FALSE;
            _arranged := TRUE;
            RETURN;
        END_IF;

        _sut.Axis_1.MoveAbsolute(inPosition := _positionAxis1,
            inVelocity := _velocity,
            inAcceleration := _acceleration,
            inDeceleration := _deceleration,
            inJerk := _jerk);

        _sut.Axis_2.MoveAbsolute(inPosition := _positionAxis2,
            inVelocity := _velocity,
            inAcceleration := _acceleration,
            inDeceleration := _deceleration,
            inJerk := _jerk);

        _sut.Axis_3.MoveAbsolute(inPosition := _positionAxis3,
            inVelocity := _velocity,
            inAcceleration := _acceleration,
            inDeceleration := _deceleration,
            inJerk := _jerk);

        _sut.Axis_4.MoveAbsolute(inPosition := _positionAxis4,
            inVelocity := _velocity,
            inAcceleration := _acceleration,
            inDeceleration := _deceleration,
            inJerk := _jerk);

        _done := (_sut.Axis_1.MoveAbsoluteTask.Done OR _sut.Axis_1.MoveAbsoluteTask.Error) AND
            (_sut.Axis_2.MoveAbsoluteTask.Done OR _sut.Axis_2.MoveAbsoluteTask.Error) AND
            (_sut.Axis_3.MoveAbsoluteTask.Done OR _sut.Axis_3.MoveAbsoluteTask.Error) AND
            (_sut.Axis_4.MoveAbsoluteTask.Done OR _sut.Axis_4.MoveAbsoluteTask.Error);

        ProbeDoneWhen(_done);
        {endregion}
        {region "T021_MoveAbsoluteEnabledNegativeDirection"}
    eTcoMultiAxisTests.MoveAbsoluteEnabledNegativeDirection:
        IF NOT _arranged THEN
            _enable := TRUE;
            _enablePositive := FALSE;
            _enableNegative := TRUE;
            _arranged := TRUE;
            RETURN;
        END_IF;

        _sut.Axis_1.MoveAbsolute(inPosition := _positionAxis1,
            inVelocity := _velocity,
            inAcceleration := _acceleration,
            inDeceleration := _deceleration,
            inJerk := _jerk);

        _sut.Axis_2.MoveAbsolute(inPosition := _positionAxis2,
            inVelocity := _velocity,
            inAcceleration := _acceleration,
            inDeceleration := _deceleration,
            inJerk := _jerk);

        _sut.Axis_3.MoveAbsolute(inPosition := _positionAxis3,
            inVelocity := _velocity,
            inAcceleration := _acceleration,
            inDeceleration := _deceleration,
            inJerk := _jerk);

        _sut.Axis_4.MoveAbsolute(inPosition := _positionAxis4,
            inVelocity := _velocity,
            inAcceleration := _acceleration,
            inDeceleration := _deceleration,
            inJerk := _jerk);

        _done := (_sut.Axis_1.MoveAbsoluteTask.Done OR _sut.Axis_1.MoveAbsoluteTask.Error) AND
            (_sut.Axis_2.MoveAbsoluteTask.Done OR _sut.Axis_2.MoveAbsoluteTask.Error) AND
            (_sut.Axis_3.MoveAbsoluteTask.Done OR _sut.Axis_3.MoveAbsoluteTask.Error) AND
            (_sut.Axis_4.MoveAbsoluteTask.Done OR _sut.Axis_4.MoveAbsoluteTask.Error);

        ProbeDoneWhen(_done);
        {endregion}
        {region "T022_MoveAbsoluteAxisDisabled"}
    eTcoMultiAxisTests.MoveAbsoluteAxisDisabled:
        IF NOT _arranged THEN
            _enable := FALSE;
            _enablePositive := FALSE;
            _enableNegative := FALSE;
            _arranged := TRUE;
            RETURN;
        END_IF;

        _moveParam.Axis1.Position := _positionAxis1;
        _moveParam.Axis1.Velocity := _velocity;
        _moveParam.Axis1.Acceleration := _acceleration;
        _moveParam.Axis1.Deceleration := _deceleration;
        _moveParam.Axis1.Jerk := _jerk;
        _moveParam.Axis2.Position := _positionAxis2;
        _moveParam.Axis2.Velocity := _velocity;
        _moveParam.Axis2.Acceleration := _acceleration;
        _moveParam.Axis2.Deceleration := _deceleration;
        _moveParam.Axis2.Jerk := _jerk;
        _moveParam.Axis3.Position := _positionAxis3;
        _moveParam.Axis3.Velocity := _velocity;
        _moveParam.Axis3.Acceleration := _acceleration;
        _moveParam.Axis3.Deceleration := _deceleration;
        _moveParam.Axis3.Jerk := _jerk;
        _moveParam.Axis4.Position := _positionAxis4;
        _moveParam.Axis4.Velocity := _velocity;
        _moveParam.Axis4.Acceleration := _acceleration;
        _moveParam.Axis4.Deceleration := _deceleration;
        _moveParam.Axis4.Jerk := _jerk;
        _sut.MoveAbsolute(_moveParam);

        _done := (_sut.MoveAbsoluteTask.Done OR _sut.MoveAbsoluteTask.Error OR _plcCycleCounter > 10) AND
            (_sut.MoveAbsoluteTask.Done OR _sut.MoveAbsoluteTask.Error OR _plcCycleCounter > 10) AND
            (_sut.MoveAbsoluteTask.Done OR _sut.MoveAbsoluteTask.Error OR _plcCycleCounter > 10) AND
            (_sut.MoveAbsoluteTask.Done OR _sut.MoveAbsoluteTask.Error OR _plcCycleCounter > 10);

        ProbeDoneWhen(_done);
        {endregion}
        {region "T023_MoveAbsoluteAxisDisabledPositiveDirection"}
    eTcoMultiAxisTests.MoveAbsoluteAxisDisabledPositiveDirection:
        IF NOT _arranged THEN
            _enable := TRUE;
            _enablePositive := FALSE;
            _enableNegative := TRUE;
            _arranged := TRUE;
            RETURN;
        END_IF;

        _moveParam.Axis1.Position := _positionAxis1;
        _moveParam.Axis1.Velocity := _velocity;
        _moveParam.Axis1.Acceleration := _acceleration;
        _moveParam.Axis1.Deceleration := _deceleration;
        _moveParam.Axis1.Jerk := _jerk;
        _moveParam.Axis2.Position := _positionAxis2;
        _moveParam.Axis2.Velocity := _velocity;
        _moveParam.Axis2.Acceleration := _acceleration;
        _moveParam.Axis2.Deceleration := _deceleration;
        _moveParam.Axis2.Jerk := _jerk;
        _moveParam.Axis3.Position := _positionAxis3;
        _moveParam.Axis3.Velocity := _velocity;
        _moveParam.Axis3.Acceleration := _acceleration;
        _moveParam.Axis3.Deceleration := _deceleration;
        _moveParam.Axis3.Jerk := _jerk;
        _moveParam.Axis4.Position := _positionAxis4;
        _moveParam.Axis4.Velocity := _velocity;
        _moveParam.Axis4.Acceleration := _acceleration;
        _moveParam.Axis4.Deceleration := _deceleration;
        _moveParam.Axis4.Jerk := _jerk;
        _sut.MoveAbsolute(_moveParam);

        _done := (_sut.MoveAbsoluteTask.Done OR (_sut.Axis_1.MoveAbsoluteTask.Error AND _sut.MoveAbsoluteTask.Error)) AND
            (_sut.MoveAbsoluteTask.Done OR (_sut.Axis_2.MoveAbsoluteTask.Error AND _sut.MoveAbsoluteTask.Error)) AND
            (_sut.MoveAbsoluteTask.Done OR (_sut.Axis_3.MoveAbsoluteTask.Error AND _sut.MoveAbsoluteTask.Error)) AND
            (_sut.MoveAbsoluteTask.Done OR (_sut.Axis_4.MoveAbsoluteTask.Error AND _sut.MoveAbsoluteTask.Error));

        ProbeDoneWhen(_done);
        {endregion}
        {region "T024_MoveAbsoluteAxisEnabledPositiveDirection"}
    eTcoMultiAxisTests.MoveAbsoluteAxisEnabledPositiveDirection:
        IF NOT _arranged THEN
            _enable := TRUE;
            _enablePositive := TRUE;
            _enableNegative := FALSE;
            _arranged := TRUE;
            RETURN;
        END_IF;

        _moveParam.Axis1.Position := _positionAxis1;
        _moveParam.Axis1.Velocity := _velocity;
        _moveParam.Axis1.Acceleration := _acceleration;
        _moveParam.Axis1.Deceleration := _deceleration;
        _moveParam.Axis1.Jerk := _jerk;
        _moveParam.Axis2.Position := _positionAxis2;
        _moveParam.Axis2.Velocity := _velocity;
        _moveParam.Axis2.Acceleration := _acceleration;
        _moveParam.Axis2.Deceleration := _deceleration;
        _moveParam.Axis2.Jerk := _jerk;
        _moveParam.Axis3.Position := _positionAxis3;
        _moveParam.Axis3.Velocity := _velocity;
        _moveParam.Axis3.Acceleration := _acceleration;
        _moveParam.Axis3.Deceleration := _deceleration;
        _moveParam.Axis3.Jerk := _jerk;
        _moveParam.Axis4.Position := _positionAxis4;
        _moveParam.Axis4.Velocity := _velocity;
        _moveParam.Axis4.Acceleration := _acceleration;
        _moveParam.Axis4.Deceleration := _deceleration;
        _moveParam.Axis4.Jerk := _jerk;
        _sut.MoveAbsolute(_moveParam);

        _done := (_sut.MoveAbsoluteTask.Done OR (_sut.Axis_1.MoveAbsoluteTask.Error AND _sut.MoveAbsoluteTask.Error)) AND
            (_sut.MoveAbsoluteTask.Done OR (_sut.Axis_2.MoveAbsoluteTask.Error AND _sut.MoveAbsoluteTask.Error)) AND
            (_sut.MoveAbsoluteTask.Done OR (_sut.Axis_3.MoveAbsoluteTask.Error AND _sut.MoveAbsoluteTask.Error)) AND
            (_sut.MoveAbsoluteTask.Done OR (_sut.Axis_4.MoveAbsoluteTask.Error AND _sut.MoveAbsoluteTask.Error));

        ProbeDoneWhen(_done);
        {endregion}
        {region "T025_MoveAbsoluteAxisDisabledNegativeDirection"}
    eTcoMultiAxisTests.MoveAbsoluteAxisDisabledNegativeDirection:
        IF NOT _arranged THEN
            _enable := TRUE;
            _enablePositive := FALSE;
            _enableNegative := FALSE;
            _arranged := TRUE;
            RETURN;
        END_IF;

        _moveParam.Axis1.Position := _positionAxis1;
        _moveParam.Axis1.Velocity := _velocity;
        _moveParam.Axis1.Acceleration := _acceleration;
        _moveParam.Axis1.Deceleration := _deceleration;
        _moveParam.Axis1.Jerk := _jerk;
        _moveParam.Axis2.Position := _positionAxis2;
        _moveParam.Axis2.Velocity := _velocity;
        _moveParam.Axis2.Acceleration := _acceleration;
        _moveParam.Axis2.Deceleration := _deceleration;
        _moveParam.Axis2.Jerk := _jerk;
        _moveParam.Axis3.Position := _positionAxis3;
        _moveParam.Axis3.Velocity := _velocity;
        _moveParam.Axis3.Acceleration := _acceleration;
        _moveParam.Axis3.Deceleration := _deceleration;
        _moveParam.Axis3.Jerk := _jerk;
        _moveParam.Axis4.Position := _positionAxis4;
        _moveParam.Axis4.Velocity := _velocity;
        _moveParam.Axis4.Acceleration := _acceleration;
        _moveParam.Axis4.Deceleration := _deceleration;
        _moveParam.Axis4.Jerk := _jerk;
        _sut.MoveAbsolute(_moveParam);

        _done := (_sut.MoveAbsoluteTask.Done OR (_sut.Axis_1.MoveAbsoluteTask.Error AND _sut.MoveAbsoluteTask.Error)) AND
            (_sut.MoveAbsoluteTask.Done OR (_sut.Axis_2.MoveAbsoluteTask.Error AND _sut.MoveAbsoluteTask.Error)) AND
            (_sut.MoveAbsoluteTask.Done OR (_sut.Axis_3.MoveAbsoluteTask.Error AND _sut.MoveAbsoluteTask.Error)) AND
            (_sut.MoveAbsoluteTask.Done OR (_sut.Axis_4.MoveAbsoluteTask.Error AND _sut.MoveAbsoluteTask.Error));

        ProbeDoneWhen(_done);
        {endregion}
        {region "T026_MoveAbsoluteAxisEnabledNegativeDirection"}
    eTcoMultiAxisTests.MoveAbsoluteAxisEnabledNegativeDirection:
        IF NOT _arranged THEN
            _enable := TRUE;
            _enablePositive := FALSE;
            _enableNegative := TRUE;
            _arranged := TRUE;
            RETURN;
        END_IF;

        _moveParam.Axis1.Position := _positionAxis1;
        _moveParam.Axis1.Velocity := _velocity;
        _moveParam.Axis1.Acceleration := _acceleration;
        _moveParam.Axis1.Deceleration := _deceleration;
        _moveParam.Axis1.Jerk := _jerk;
        _moveParam.Axis2.Position := _positionAxis2;
        _moveParam.Axis2.Velocity := _velocity;
        _moveParam.Axis2.Acceleration := _acceleration;
        _moveParam.Axis2.Deceleration := _deceleration;
        _moveParam.Axis2.Jerk := _jerk;
        _moveParam.Axis3.Position := _positionAxis3;
        _moveParam.Axis3.Velocity := _velocity;
        _moveParam.Axis3.Acceleration := _acceleration;
        _moveParam.Axis3.Deceleration := _deceleration;
        _moveParam.Axis3.Jerk := _jerk;
        _moveParam.Axis4.Position := _positionAxis4;
        _moveParam.Axis4.Velocity := _velocity;
        _moveParam.Axis4.Acceleration := _acceleration;
        _moveParam.Axis4.Deceleration := _deceleration;
        _moveParam.Axis4.Jerk := _jerk;
        _sut.MoveAbsolute(_moveParam);

        _done := (_sut.MoveAbsoluteTask.Done OR (_sut.Axis_1.MoveAbsoluteTask.Error AND _sut.MoveAbsoluteTask.Error)) AND
            (_sut.MoveAbsoluteTask.Done OR (_sut.Axis_2.MoveAbsoluteTask.Error AND _sut.MoveAbsoluteTask.Error)) AND
            (_sut.MoveAbsoluteTask.Done OR (_sut.Axis_3.MoveAbsoluteTask.Error AND _sut.MoveAbsoluteTask.Error)) AND
            (_sut.MoveAbsoluteTask.Done OR (_sut.Axis_4.MoveAbsoluteTask.Error AND _sut.MoveAbsoluteTask.Error));

        ProbeDoneWhen(_done);
        {endregion}
        {region "T027_MoveAbsoluteAxisDisabledPositiveDirectionAxisDisabled"}
    eTcoMultiAxisTests.MoveAbsoluteAxisDisabledPositiveDirectionAxisDisabled:
        IF NOT _arranged THEN
            _enable := TRUE;
            _enablePositive := FALSE;
            _enableNegative := TRUE;
            _arranged := TRUE;
            RETURN;
        END_IF;

        _moveParam.Axis1.Position := _positionAxis1;
        _moveParam.Axis1.Velocity := _velocity;
        _moveParam.Axis1.Acceleration := _acceleration;
        _moveParam.Axis1.Deceleration := _deceleration;
        _moveParam.Axis1.Jerk := _jerk;
        _moveParam.Axis2.Position := _positionAxis2;
        _moveParam.Axis2.Velocity := _velocity;
        _moveParam.Axis2.Acceleration := _acceleration;
        _moveParam.Axis2.Deceleration := _deceleration;
        _moveParam.Axis2.Jerk := _jerk;
        _moveParam.Axis3.Position := _positionAxis3;
        _moveParam.Axis3.Velocity := _velocity;
        _moveParam.Axis3.Acceleration := _acceleration;
        _moveParam.Axis3.Deceleration := _deceleration;
        _moveParam.Axis3.Jerk := _jerk;
        _moveParam.Axis4.Position := _positionAxis4;
        _moveParam.Axis4.Velocity := _velocity;
        _moveParam.Axis4.Acceleration := _acceleration;
        _moveParam.Axis4.Deceleration := _deceleration;
        _moveParam.Axis4.Jerk := _jerk;
        _sut.MoveAbsolute(_moveParam);
        _done := _sut.MoveAbsoluteTask.Done OR _sut.MoveAbsoluteTask.Error;
        ProbeDoneWhen(_done);
        {endregion}
        {region "T028_MoveAbsoluteAxisEnabledPositiveDirectionAxisDisabled"}
    eTcoMultiAxisTests.MoveAbsoluteAxisEnabledPositiveDirectionAxisDisabled:
        IF NOT _arranged THEN
            _enable := TRUE;
            _enablePositive := TRUE;
            _enableNegative := FALSE;
            _arranged := TRUE;
            RETURN;
        END_IF;

        _moveParam.Axis1.Position := _positionAxis1;
        _moveParam.Axis1.Velocity := _velocity;
        _moveParam.Axis1.Acceleration := _acceleration;
        _moveParam.Axis1.Deceleration := _deceleration;
        _moveParam.Axis1.Jerk := _jerk;
        _moveParam.Axis2.Position := _positionAxis2;
        _moveParam.Axis2.Velocity := _velocity;
        _moveParam.Axis2.Acceleration := _acceleration;
        _moveParam.Axis2.Deceleration := _deceleration;
        _moveParam.Axis2.Jerk := _jerk;
        _moveParam.Axis3.Position := _positionAxis3;
        _moveParam.Axis3.Velocity := _velocity;
        _moveParam.Axis3.Acceleration := _acceleration;
        _moveParam.Axis3.Deceleration := _deceleration;
        _moveParam.Axis3.Jerk := _jerk;
        _moveParam.Axis4.Position := _positionAxis4;
        _moveParam.Axis4.Velocity := _velocity;
        _moveParam.Axis4.Acceleration := _acceleration;
        _moveParam.Axis4.Deceleration := _deceleration;
        _moveParam.Axis4.Jerk := _jerk;
        _sut.MoveAbsolute(_moveParam);
        _done := _sut.MoveAbsoluteTask.Done OR _sut.MoveAbsoluteTask.Error;
        ProbeDoneWhen(_done);
        {region "T029_MoveAbsoluteAxisDisabledNegativeDirectionAxisDisabled"}
    eTcoMultiAxisTests.MoveAbsoluteAxisDisabledNegativeDirectionAxisDisabled:
        IF NOT _arranged THEN
            _enable := TRUE;
            _enablePositive := FALSE;
            _enableNegative := FALSE;
            _arranged := TRUE;
            RETURN;
        END_IF;

        _moveParam.Axis1.Position := _positionAxis1;
        _moveParam.Axis1.Velocity := _velocity;
        _moveParam.Axis1.Acceleration := _acceleration;
        _moveParam.Axis1.Deceleration := _deceleration;
        _moveParam.Axis1.Jerk := _jerk;
        _moveParam.Axis2.Position := _positionAxis2;
        _moveParam.Axis2.Velocity := _velocity;
        _moveParam.Axis2.Acceleration := _acceleration;
        _moveParam.Axis2.Deceleration := _deceleration;
        _moveParam.Axis2.Jerk := _jerk;
        _moveParam.Axis3.Position := _positionAxis3;
        _moveParam.Axis3.Velocity := _velocity;
        _moveParam.Axis3.Acceleration := _acceleration;
        _moveParam.Axis3.Deceleration := _deceleration;
        _moveParam.Axis3.Jerk := _jerk;
        _moveParam.Axis4.Position := _positionAxis4;
        _moveParam.Axis4.Velocity := _velocity;
        _moveParam.Axis4.Acceleration := _acceleration;
        _moveParam.Axis4.Deceleration := _deceleration;
        _moveParam.Axis4.Jerk := _jerk;
        _sut.MoveAbsolute(_moveParam);
        _done := _sut.MoveAbsoluteTask.Done OR _sut.MoveAbsoluteTask.Error;
        ProbeDoneWhen(_done);
        {endregion}
        {region "T030_MoveAbsoluteAxisEnabledNegativeDirectionAxisDisabled"}
    eTcoMultiAxisTests.MoveAbsoluteAxisEnabledNegativeDirectionAxisDisabled:
        IF NOT _arranged THEN
            _enable := TRUE;
            _enablePositive := FALSE;
            _enableNegative := TRUE;
            _arranged := TRUE;
            RETURN;
        END_IF;

        _moveParam.Axis1.Position := _positionAxis1;
        _moveParam.Axis1.Velocity := _velocity;
        _moveParam.Axis1.Acceleration := _acceleration;
        _moveParam.Axis1.Deceleration := _deceleration;
        _moveParam.Axis1.Jerk := _jerk;
        _moveParam.Axis2.Position := _positionAxis2;
        _moveParam.Axis2.Velocity := _velocity;
        _moveParam.Axis2.Acceleration := _acceleration;
        _moveParam.Axis2.Deceleration := _deceleration;
        _moveParam.Axis2.Jerk := _jerk;
        _moveParam.Axis3.Position := _positionAxis3;
        _moveParam.Axis3.Velocity := _velocity;
        _moveParam.Axis3.Acceleration := _acceleration;
        _moveParam.Axis3.Deceleration := _deceleration;
        _moveParam.Axis3.Jerk := _jerk;
        _moveParam.Axis4.Position := _positionAxis4;
        _moveParam.Axis4.Velocity := _velocity;
        _moveParam.Axis4.Acceleration := _acceleration;
        _moveParam.Axis4.Deceleration := _deceleration;
        _moveParam.Axis4.Jerk := _jerk;
        _sut.MoveAbsolute(_moveParam);
        _done := _sut.MoveAbsoluteTask.Done OR _sut.MoveAbsoluteTask.Error;
        ProbeDoneWhen(_done);
        {endregion}
END_CASE
END_METHOD

END_FUNCTION_BLOCK

// ---- Tests/TcoMultiAxis/TcoMultiAxisTest.TcPOU
FUNCTION_BLOCK TcoMultiAxisTest EXTENDS TcoDrivesBeckhoff.TcoMultiAxis
VAR
    _serviceModeCount : ULINT;
    _serviceModeOverride : LREAL;
    inoPosition : TcoMultiAxisPositionsRootContainer(THIS^);
END_VAR
VAR
    _MC_ReadDriveAddress : MC_ReadDriveAddress;
    _fbEcCoeSdoRead : FB_EcCoeSdoRead;
    sNetId : T_AmsNetId;
    nSlaveAddr : UINT;
    _MotorType : STRING;
    _ftrig : Tc2_Standard.F_TRIG;
    _MC_ReadParameter : MC_ReadParameter;
END_VAR

SUPER^(inEnableAxis1 := inEnableAxis1,
    inEnablePositiveAxis1 := inEnablePositiveAxis1,
    inEnableNegativeAxis1 := inEnableNegativeAxis1,
    inCalibrationCamAxis1 := inCalibrationCamAxis1,
    refAxis1 := refAxis1,
    inEnableAxis2 := inEnableAxis2,
    inEnablePositiveAxis2 := inEnablePositiveAxis2,
    inEnableNegativeAxis2 := inEnableNegativeAxis2,
    inCalibrationCamAxis2 := inCalibrationCamAxis2,
    refAxis2 := refAxis2,
    inEnableAxis3 := inEnableAxis3,
    inEnablePositiveAxis3 := inEnablePositiveAxis3,
    inEnableNegativeAxis3 := inEnableNegativeAxis3,
    inCalibrationCamAxis3 := inCalibrationCamAxis3,
    refAxis3 := refAxis3,
    inEnableAxis3 := inEnableAxis4,
    inEnablePositiveAxis4 := inEnablePositiveAxis4,
    inEnableNegativeAxis4 := inEnableNegativeAxis4,
    inCalibrationCamAxis4 := inCalibrationCamAxis4,
    refAxis4 := refAxis4,
    inoPositions := inoPosition);

END_FUNCTION_BLOCK

// ---- Tests/TcoContext/SomeTestMultiPositions.TcPOU
FUNCTION_BLOCK SomeTestMultiPositions EXTENDS TcoDrivesBeckhoff.TcoMultiAxisPositionsRootContainer
VAR_INPUT
END_VAR
VAR_OUTPUT
END_VAR
VAR
    {attribute addProperty Name "<#Pick Position#>"}
    PickPosition : TcoDrivesBeckhoff.TcoMultiAxisMoveParam;
    {attribute addProperty Name "<#Place  Position#>"}
    PlacePosition : TcoDrivesBeckhoff.TcoMultiAxisMoveParam;
END_VAR

PROPERTY PUBLIC PickPos : REFERENCE TO TcoDrivesBeckhoff.TcoMultiAxisMoveParam;
GET
PickPos REF= PickPosition;
END_GET
END_PROPERTY

PROPERTY PUBLIC PlacePos : REFERENCE TO TcoDrivesBeckhoff.TcoMultiAxisMoveParam;
GET
PlacePos REF= PlacePosition;
END_GET
END_PROPERTY

END_FUNCTION_BLOCK

// ---- Tests/TcoContext/WpfContext.TcPOU
FUNCTION_BLOCK WpfContext EXTENDS TcoCore.TcoContext
VAR
    _serviceModeActive : BOOL;
    {attribute addProperty Name "<#Test axis 1#>"}
    _axis1 : TcoDrivesBeckhoff.TcoDriveSimple(THIS^);
    _enable1 : BOOL;
    _enablePositive1 : BOOL;
    _enableNegative1 : BOOL;
    _calibrationCam1 : BOOL;
    {attribute addProperty Name "<#Test axis 2#>"}
    _axis2 : TcoDrivesBeckhoff.TcoDriveSimple(THIS^);
    _enable2 : BOOL;
    _enablePositive2 : BOOL;
    _enableNegative2 : BOOL;
    _calibrationCam2 : BOOL;
    _enableMulti : BOOL;
    _enableMultiPositive : BOOL;
    _enableMultiNegative : BOOL;
    _calibrationMultiCam : BOOL;
    {attribute addProperty Name "<#Test positions#>"}
    _positions : SomeTestPositions(THIS^);
    {attribute addProperty Name "<#Test single axis#>"}
    _singleAxis : TcoDrivesBeckhoff.TcoSingleAxis(THIS^);
    {attribute addProperty Name "<#Test multi positions#>"}
    _positionsMulti : SomeTestMultiPositions(THIS^);
    {attribute addProperty Name "<#Test multi axis#>"}
    _multiAxis : TcoDrivesBeckhoff.TcoMultiAxis(THIS^);
    {attribute addProperty Name "<#Wrapped Component Example#>"}
    _wrappedExample : WrappedComponentExample(THIS^);
    _sequence1 : TcoCore.TcoSequence(THIS^, eRestoreMode.None);
    _observer : TcoCore.TcoSequencerObserver(THIS^);
    {attribute addProperty Name "Start sequence"}
    _sequence1Task : Sequence1Task(THIS^);
    _dialog : TcoCore.TcoDialog(THIS^);
    _moveParam : TcoMultiAxisMoveParam;
END_VAR

(*~
    <docu>
        <summary>
            Main method of the TcoContext. This is the entry point of any control logic that belongs to this context.
            The call of this method is ensured by calling the <c>InstanceName.Run()</c> method, and it must not be called explicitly.
            This method is abstract, and it must be overridden in derived block.
        </summary>
    </docu>
~*)
METHOD PROTECTED Main
IF _serviceModeActive THEN
    _axis1.Service();
    _axis2.Service();
    _singleAxis.Service();
    _multiAxis.Service();
END_IF

_axis1(inEnable := _enable1,
    inEnablePositive := _enablePositive1,
    inEnableNegative := _enableNegative1,
    inCalibrationCam := _calibrationCam1 or GVL._calibrationCam,
    inoAxisRef := GVL.SimpleAxis1);

_axis2(inEnable := _enable2,
    inEnablePositive := _enablePositive2,
    inEnableNegative := _enableNegative2,
    inCalibrationCam := _calibrationCam2,
    inoAxisRef := GVL.SimpleAxis2);

_singleAxis.Config.InfoTime := T#4S;
_singleAxis.Config.ErrorTime := T#10S;
//example how to permanently disable(hide in service view)not required functionalities(or can be defined as settable parameters)
_singleAxis.Axis.Config.HideHalt := TRUE;

_singleAxis(inEnable := _enable1,
    inEnablePositive := _enablePositive1,
    inEnableNegative := _enableNegative1,
    inCalibrationCam := _calibrationCam1 or GVL._calibrationCam,
    refAxis := GVL.SingleAxis,
    inoPositions := _positions);
// this means it is three axis cartesian system
//_multiAxis.Config.Axis4Disabled:=TRUE;
_multiAxis.Config.InfoTime := T#4S;
_multiAxis.Config.ErrorTime := T#10S;
//example how to permanently disable(hide in service view)not required functionalities(or can be defined as settable parameters)
_multiAxis.Axis_1.Config.HideHalt := TRUE;

_multiAxis(inEnableAxis1 := _enableMulti,
    inEnablePositiveAxis1 := _enableMultiPositive,
    inEnableNegativeAxis1 := _enableMultiNegative,
    inCalibrationCamAxis1 := _calibrationMultiCam OR GVL._calibrationCam,
    refAxis1 := GVL.Axis1,
    inEnableAxis2 := _enableMulti,
    inEnablePositiveAxis2 := _enableMultiPositive,
    inEnableNegativeAxis2 := _enableMultiNegative,
    inCalibrationCamAxis2 := _calibrationMultiCam OR GVL._calibrationCam,
    refAxis2 := GVL.Axis2,
    inEnableAxis3 := _enableMulti,
    inEnablePositiveAxis3 := _enableMultiPositive,
    inEnableNegativeAxis3 := _enableMultiNegative,
    inCalibrationCamAxis3 := _calibrationMultiCam OR GVL._calibrationCam,
    refAxis3 := GVL.Axis3,
    inEnableAxis4 := _enableMulti,
    inEnablePositiveAxis4 := _enableMultiPositive,
    inEnableNegativeAxis4 := _enableMultiNegative,
    inCalibrationCamAxis4 := _calibrationMultiCam OR GVL._calibrationCam,
    refAxis4 := GVL.Axis4,
    inoPositions := _positionsMulti);

_sequence1Task(Sequence := _sequence1);

IF (_sequence1Task.Execute()) THEN
    Sequence1();
END_IF;
END_METHOD

METHOD Sequence1
VAR
    seq : REFERENCE TO TcoCore.TcoSequence;
    answer : TcoCore.eDialogAnswer;
    done : BOOL;
    _jerk : LREAL;
    _deceleration : LREAL;
    _acceleration : LREAL;
    _velocity : LREAL;
    ProbeDoneWhen : INT;
END_VAR
seq REF= _sequence1;
seq.Open();
seq.Observer := _observer;

IF (seq.Step(inStepID := 0, inEnabled := TRUE, inStepDescription := 'READY TO START')) THEN
    //--------------------------------------------------------
    answer := _dialog.Show()
        .WithType(eDialogType.Question)
        .WithCaption('Ready to go?')
        .WithText('Do you really want to start movements? Do we go ahead?')
        .WithYesNo().Answer;

    //
    IF (answer = TcoCore.eDialogAnswer.Yes) THEN
        seq.CompleteStep();
    ELSIF (answer = TcoCore.eDialogAnswer.No) THEN
        _sequence1Task.Restore();
    END_IF;
    //--------------------------------------------------------
END_IF;

IF (seq.Step(inStepID := 10, inEnabled := TRUE, inStepDescription := 'MULTI AXIS  HOMING IF NECESSARY')) THEN
    //--------------------------------------------------------
    _enableMulti := TRUE;
    _enableMultiNegative := TRUE;
    _enableMultiPositive := TRUE;

    IF _multiAxis.Axis_1._axisStatus.Operational AND
        _multiAxis.Axis_1._axisStatus.Homed AND
        _multiAxis.Axis_2._axisStatus.Operational AND
        _multiAxis.Axis_2._axisStatus.Homed AND
        _multiAxis.Axis_3._axisStatus.Operational AND
        _multiAxis.Axis_3._axisStatus.Homed AND
        _multiAxis.Axis_4._axisStatus.Operational AND
        _multiAxis.Axis_4._axisStatus.Homed THEN
        seq.CompleteStep();
    ELSIF _multiAxis.Axis_1._axisStatus.Operational AND
        _multiAxis.Axis_2._axisStatus.Operational AND
        _multiAxis.Axis_3._axisStatus.Operational AND
        _multiAxis.Axis_4._axisStatus.Operational THEN
        _multiAxis.Axis_1.Home(inPosition := 0,
            inHomingMode := TcoDrivesBeckhoff.eHomingMode.MC_Direct,
            inClearPositionLag := FALSE,
            inSearchDirection := TcoDrivesBeckhoff.eDirection.MC_Undefined_Direction,
            inSearchVelocity := _velocity,
            inSyncDirection := TcoDrivesBeckhoff.eDirection.MC_Undefined_Direction,
            inSyncVelocity := _velocity,
            inReferenceMode := TcoDrivesBeckhoff.eEncoderReferenceMode.ENCODERREFERENCEMODE_DEFAULT);

        _multiAxis.Axis_2.Home(inPosition := 0,
            inHomingMode := TcoDrivesBeckhoff.eHomingMode.MC_Direct,
            inClearPositionLag := FALSE,
            inSearchDirection := TcoDrivesBeckhoff.eDirection.MC_Undefined_Direction,
            inSearchVelocity := _velocity,
            inSyncDirection := TcoDrivesBeckhoff.eDirection.MC_Undefined_Direction,
            inSyncVelocity := _velocity,
            inReferenceMode := TcoDrivesBeckhoff.eEncoderReferenceMode.ENCODERREFERENCEMODE_DEFAULT);

        _multiAxis.Axis_3.Home(inPosition := 0,
            inHomingMode := TcoDrivesBeckhoff.eHomingMode.MC_Direct,
            inClearPositionLag := FALSE,
            inSearchDirection := TcoDrivesBeckhoff.eDirection.MC_Undefined_Direction,
            inSearchVelocity := _velocity,
            inSyncDirection := TcoDrivesBeckhoff.eDirection.MC_Undefined_Direction,
            inSyncVelocity := _velocity,
            inReferenceMode := TcoDrivesBeckhoff.eEncoderReferenceMode.ENCODERREFERENCEMODE_DEFAULT);

        _multiAxis.Axis_4.Home(inPosition := 0,
            inHomingMode := TcoDrivesBeckhoff.eHomingMode.MC_Direct,
            inClearPositionLag := FALSE,
            inSearchDirection := TcoDrivesBeckhoff.eDirection.MC_Undefined_Direction,
            inSearchVelocity := _velocity,
            inSyncDirection := TcoDrivesBeckhoff.eDirection.MC_Undefined_Direction,
            inSyncVelocity := _velocity,
            inReferenceMode := TcoDrivesBeckhoff.eEncoderReferenceMode.ENCODERREFERENCEMODE_DEFAULT);

        IF (_multiAxis.Axis_1.HomeTask.Done OR _multiAxis.Axis_1.HomeTask.Error) AND
            (_multiAxis.Axis_2.HomeTask.Done OR _multiAxis.Axis_2.HomeTask.Error) AND
            (_multiAxis.Axis_3.HomeTask.Done OR _multiAxis.Axis_3.HomeTask.Error) AND
            (_multiAxis.Axis_4.HomeTask.Done OR _multiAxis.Axis_4.HomeTask.Error) THEN
            seq.CompleteStep();
        END_IF;
    ELSE
        answer := _dialog.Show()
            .WithType(eDialogType.Question)
            .WithCaption('SOME ERROR')
            .WithText('There are some errors, restore will be provided!')
            .WithOk().Answer;

        IF (answer = TcoCore.eDialogAnswer.OK) THEN
            _multiAxis.Restore();
            _sequence1Task.Restore();
        END_IF;
    END_IF;
    //--------------------------------------------------------
END_IF;

IF (seq.Step(inStepID := 11, inEnabled := TRUE, inStepDescription := 'LOAD POSITIONS')) THEN
    //--------------------------------------------------------
    IF _multiAxis.LoadPositionsTask.WithId('default').Invoke().Done THEN
        seq.CompleteStep();
    END_IF

    //--------------------------------------------------------
END_IF;

IF (seq.Step(inStepID := 12, inEnabled := _multiAxis.LoadPositionsTask.DoesNotExist, inStepDescription := 'LOAD/CREATE POSITIONS')) THEN
    //--------------------------------------------------------
    answer := _dialog.Show()
        .WithType(eDialogType.Question)
        .WithCaption('Positions set missing!')
        .WithText('Do you really want create default set?')
        .WithYesNo().Answer;

    //
    IF (answer = TcoCore.eDialogAnswer.Yes) THEN
        seq.CompleteStep();
    ELSIF (answer = TcoCore.eDialogAnswer.No) THEN
        _sequence1Task.Restore();
    END_IF;
    //--------------------------------------------------------
END_IF;

IF (seq.Step(inStepID := 13,
    inEnabled := _multiAxis.LoadPositionsTask.DoesNotExist,
    inStepDescription := 'POSITION NOT EXIST NECESSARY TO CREATE POSITIONS')) THEN
    //--------------------------------------------------------
    _velocity := 1400;
    _deceleration := 5000;
    _acceleration := 5000;
    _jerk := 15000;
    _positionsMulti.PickPos.Axis1.Position := _multiAxis.Axis_1.AxisStatus.ActPos - 1000;
    _positionsMulti.PickPos.Axis1.Velocity := _velocity;
    _positionsMulti.PickPos.Axis1.Acceleration := _acceleration;
    _positionsMulti.PickPos.Axis1.Deceleration := _deceleration;
    _positionsMulti.PickPos.Axis1.Jerk := _jerk;
    _positionsMulti.PickPos.Axis2.Position := _multiAxis.Axis_2.AxisStatus.ActPos - 1000;
    _positionsMulti.PickPos.Axis2.Velocity := _velocity;
    _positionsMulti.PickPos.Axis2.Acceleration := _acceleration;
    _positionsMulti.PickPos.Axis2.Deceleration := _deceleration;
    _positionsMulti.PickPos.Axis2.Jerk := _jerk;
    _positionsMulti.PickPos.Axis3.Position := _multiAxis.Axis_3.AxisStatus.ActPos - 1000;
    _positionsMulti.PickPos.Axis3.Velocity := _velocity;
    _positionsMulti.PickPos.Axis3.Acceleration := _acceleration;
    _positionsMulti.PickPos.Axis3.Deceleration := _deceleration;
    _positionsMulti.PickPos.Axis3.Jerk := _jerk;
    _positionsMulti.PickPos.Axis4.Position := _multiAxis.Axis_4.AxisStatus.ActPos - 1000;
    _positionsMulti.PickPos.Axis4.Velocity := _velocity;
    _positionsMulti.PickPos.Axis4.Acceleration := _acceleration;
    _positionsMulti.PickPos.Axis4.Deceleration := _deceleration;
    _positionsMulti.PickPos.Axis4.Jerk := _jerk;

    IF _multiAxis.SavePositionsTask.WithId('default').Invoke().Done AND _multiAxis.SavePositionsTask.ReadSuccessfuly THEN
        seq.CompleteStep();
    END_IF
    //--------------------------------------------------------
END_IF;

IF (seq.Step(inStepID := 14, inEnabled := TRUE, inStepDescription := 'LOAD CREATED POSITIONS')) THEN
    //--------------------------------------------------------
    IF _multiAxis.LoadPositionsTask.WithId('default').Invoke().Done AND _multiAxis.LoadPositionsTask.ReadSuccessfuly THEN
        seq.CompleteStep();
    END_IF

    //--------------------------------------------------------
END_IF

IF (seq.Step(inStepID := 25, inEnabled := TRUE, inStepDescription := 'MULTI AXIS  MOVEMENTS')) THEN
    //--------------------------------------------------------
    _enableMulti := TRUE;
    _enableMultiNegative := TRUE;
    _enableMultiPositive := TRUE;

    //
    //		_moveParam.Axis1.Position:= _multiAxis.Axis_1.AxisStatus.ActPos-1000;
    //		_moveParam.Axis1.Velocity := _velocity;
    //		_moveParam.Axis1.Acceleration := _acceleration;
    //		_moveParam.Axis1.Deceleration := _deceleration;
    //		_moveParam.Axis1.Jerk :=  _jerk;
    //
    //
    //		_moveParam.Axis2.Position:= _multiAxis.Axis_2.AxisStatus.ActPos-1000;
    //		_moveParam.Axis2.Velocity := _velocity;
    //		_moveParam.Axis2.Acceleration := _acceleration;
    //		_moveParam.Axis2.Deceleration := _deceleration;
    //		_moveParam.Axis2.Jerk :=  _jerk;
    //
    //		_moveParam.Axis3.Position:= _multiAxis.Axis_3.AxisStatus.ActPos-1000;
    //		_moveParam.Axis3.Velocity := _velocity;
    //		_moveParam.Axis3.Acceleration := _acceleration;
    //		_moveParam.Axis3.Deceleration := _deceleration;
    //		_moveParam.Axis3.Jerk :=  _jerk;
    //
    //		_moveParam.Axis4.Position:= _multiAxis.Axis_4.AxisStatus.ActPos-1000;
    //		_moveParam.Axis4.Velocity := _velocity;
    //		_moveParam.Axis4.Acceleration := _acceleration;
    //		_moveParam.Axis4.Deceleration := _deceleration;
    //		_moveParam.Axis4.Jerk :=  _jerk;
    IF _multiAxis.MoveAbsolute(_positionsMulti.PickPos).Done THEN
        seq.CompleteStep();
    END_IF
    //--------------------------------------------------------
END_IF;

IF (seq.Step(inStepID := 50, inEnabled := TRUE, inStepDescription := 'SIMULATE ERROR')) THEN
    //--------------------------------------------------------
    //<StandardDialog>
    answer :=
        _dialog.Show().WithType(eDialogType.Question).WithCaption('Question?').WithText('Do you really want to simulate error?').WithYesNo().Answer;

    //
    IF (answer = TcoCore.eDialogAnswer.Yes) THEN
        seq.CompleteStep();
    ELSIF (answer = TcoCore.eDialogAnswer.No) THEN
        _sequence1Task.Restore();
    END_IF;
    //--------------------------------------------------------
END_IF;

IF (seq.Step(inStepID := 100, inEnabled := TRUE, inStepDescription := 'MULTI AXIS SIMULATE ERROR')) THEN
    //--------------------------------------------------------
    _enableMulti := TRUE;
    _enableMultiNegative := TRUE;
    _enableMultiPositive := TRUE;
    _velocity := 15000;
    _deceleration := -1;
    _acceleration := -1;
    _jerk := 15000;
    _moveParam.Axis1.Position := _multiAxis.Axis_1.AxisStatus.ActPos - 1000;
    _moveParam.Axis1.Velocity := _velocity;
    _moveParam.Axis1.Acceleration := _acceleration;
    _moveParam.Axis1.Deceleration := _deceleration;
    _moveParam.Axis1.Jerk := _jerk;
    _moveParam.Axis2.Position := _multiAxis.Axis_2.AxisStatus.ActPos - 1000;
    _moveParam.Axis2.Velocity := _velocity;
    _moveParam.Axis2.Acceleration := _acceleration;
    _moveParam.Axis2.Deceleration := _deceleration;
    _moveParam.Axis2.Jerk := _jerk;
    _moveParam.Axis3.Position := _multiAxis.Axis_3.AxisStatus.ActPos - 1000;
    _moveParam.Axis3.Velocity := _velocity;
    _moveParam.Axis3.Acceleration := _acceleration;
    _moveParam.Axis3.Deceleration := _deceleration;
    _moveParam.Axis3.Jerk := _jerk;
    _moveParam.Axis4.Position := _multiAxis.Axis_4.AxisStatus.ActPos - 1000;
    _moveParam.Axis4.Velocity := _velocity;
    _moveParam.Axis4.Acceleration := _acceleration;
    _moveParam.Axis4.Deceleration := _deceleration;
    _moveParam.Axis4.Jerk := _jerk;

    IF _multiAxis.MoveAbsolute(_moveParam).Error THEN
        seq.CompleteStep();
    END_IF
    //--------------------------------------------------------
END_IF;

//<TcoDigitalInspector>
IF (seq.Step(inStepID := 200, inEnabled := TRUE, inStepDescription := 'CLEAR ERROR')) THEN
    //--------------------------------------------------------
    //<StandardDialog>
    answer := _dialog.Show().WithType(eDialogType.Question).WithCaption('Question?').WithText('Do you want to reset error?').WithYesNo().Answer;

    //
    IF (answer = TcoCore.eDialogAnswer.Yes) THEN
        seq.CompleteStep();
    ELSIF (answer = TcoCore.eDialogAnswer.No) THEN
        _sequence1Task.Restore();
    END_IF;
    //--------------------------------------------------------
END_IF;

IF (seq.Step(inStepID := 249, inEnabled := TRUE, inStepDescription := 'RESET AXIS')) THEN
    //--------------------------------------------------------
    IF _multiAxis.ResetDrives().Done AND_THEN
        NOT _multiAxis.Axis_1.AxisStatus.Error AND
        NOT _multiAxis.Axis_2.AxisStatus.Error AND
        NOT _multiAxis.Axis_2.AxisStatus.Error AND
        NOT _multiAxis.Axis_2.AxisStatus.Error THEN
        seq.CompleteStep();
    end_if;
    //--------------------------------------------------------
END_IF;

IF (seq.Step(inStepID := 300, inEnabled := TRUE, inStepDescription := 'ASKING FOR RESTORING')) THEN
    //--------------------------------------------------------
    //<StandardDialog>
    answer := _dialog.Show()
        .WithType(eDialogType.Question)
        .WithCaption('Question?')
        .WithText('Do you want to restore MultiAxis component?')
        .WithYesNo().Answer;

    //
    IF (answer = TcoCore.eDialogAnswer.Yes) THEN
        _multiAxis.Restore();
        seq.CompleteStep();
    ELSIF (answer = TcoCore.eDialogAnswer.No) THEN
        _sequence1Task.Restore();
    END_IF;
    //--------------------------------------------------------
END_IF;

IF (seq.Step(inStepID := 400, inEnabled := TRUE, inStepDescription := 'MOVE WITH ONLY ONE AXIS')) THEN
    //--------------------------------------------------------
    answer := _dialog.Show()
        .WithType(eDialogType.Question)
        .WithCaption('ONE AXIS EXAMPLE?')
        .WithText('Do you  want to start movements with one axis?')
        .WithYesNo().Answer;

    //
    IF (answer = TcoCore.eDialogAnswer.Yes) THEN
        seq.CompleteStep();
    ELSIF (answer = TcoCore.eDialogAnswer.No) THEN
        _sequence1Task.Restore();
    END_IF;
    //--------------------------------------------------------
END_IF;

IF (seq.Step(inStepID := 425, inEnabled := TRUE, inStepDescription := 'ONE AXIS EXAMPLE')) THEN
    //--------------------------------------------------------
    _enableMulti := TRUE;
    _enableMultiNegative := TRUE;
    _enableMultiPositive := TRUE;
    _velocity := 1400;
    _deceleration := 5000;
    _acceleration := 5000;
    _jerk := 15000;

    IF _multiAxis.Axis_1.MoveAbsolute(inPosition := _multiAxis.Axis_1.AxisStatus.ActPos - 1000,
        inVelocity := _velocity,
        inAcceleration := _acceleration,
        inDeceleration := _deceleration,
        inJerk := _jerk).Done THEN
        seq.CompleteStep();
    END_IF
    //--------------------------------------------------------
END_IF;

IF (seq.Step(inStepID := 500, inEnabled := TRUE, inStepDescription := 'EXAMPLE LONG RANGE MOVMENT ABORTED')) THEN
    //--------------------------------------------------------
    answer := _dialog.Show()
        .WithType(eDialogType.Question)
        .WithCaption('Abort movement?')
        .WithText('Do you  want to start movements and abort it?')
        .WithYesNo().Answer;

    //
    IF (answer = TcoCore.eDialogAnswer.Yes) THEN
        seq.CompleteStep();
    ELSIF (answer = TcoCore.eDialogAnswer.No) THEN
        _sequence1Task.Restore();
    END_IF;
    //--------------------------------------------------------
END_IF;

IF (seq.Step(inStepID := 525, inEnabled := TRUE, inStepDescription := 'ABORT MOVEMENT AXIS EXAMPLE')) THEN
    //--------------------------------------------------------
    _enableMulti := TRUE;
    _enableMultiNegative := TRUE;
    _enableMultiPositive := TRUE;
    _velocity := 1400;
    _deceleration := 5000;
    _acceleration := 5000;
    _jerk := 15000;

    answer :=
        _dialog.Show().WithType(eDialogType.Question).WithCaption('Movement running').WithText('Do you  want to abort movement?').WithYesNo().Answer;

    //
    IF (answer = TcoCore.eDialogAnswer.Yes) THEN
        _multiAxis.AbortTask.Invoke();
        seq.CompleteStep();
    ELSIF (answer = TcoCore.eDialogAnswer.No) THEN
        _sequence1Task.Restore();
    END_IF;

